// TIA Portal V17 program export: 2 tag tables, 13 data types, 7 data blocks, 53 code blocks (in call order from the OBs), 36 instance data blocks

VAR_GLOBAL   // PLC tag table "Default tag table"
   System_Byte AT %MB1 : Byte;
   FirstScan AT %M1.0 : Bool;
   DiagStatusUpdate AT %M1.1 : Bool;
   Clock_Byte AT %MB0 : Byte;
   Clock_10Hz AT %M0.0 : Bool;
   Clock_5Hz AT %M0.1 : Bool;
   "Clock_2.5Hz" AT %M0.2 : Bool;
   Clock_2Hz AT %M0.3 : Bool;
   "Clock_1.25Hz" AT %M0.4 : Bool;
   Clock_1Hz AT %M0.5 : Bool;
   "Clock_0.625Hz" AT %M0.6 : Bool;
   "Clock_0.5Hz" AT %M0.7 : Bool;
   "System_Byte(1)" AT %MB1 : Byte;
   AlwaysTRUE AT %M1.2 : Bool;
   AlwaysFALSE AT %M1.3 : Bool;
   "System_Byte(2)" AT %MB1 : Byte;
   Tag_1 AT %Q0.6 : Bool;
   Tag_2 AT %M110.0 : Bool;
   Tag_3 AT %M110.1 : Bool;
   Tag_4 AT %MW110 : Word;
END_VAR

VAR_GLOBAL   // PLC tag table "System_Tags"
   pulse_01s AT %M10.0 : Bool;
   pulse_05s AT %M10.1 : Bool;
   pulse_1s AT %M10.2 : Bool;
   pulse_5s AT %M10.3 : Bool;
   pulse_10s AT %M10.4 : Bool;
   pulse_30s AT %M10.5 : Bool;
   pulse_1m AT %M10.6 : Bool;
   pulse_5m AT %M10.7 : Bool;
   pulse_10m AT %M11.0 : Bool;
   pulse_1h AT %M11.2 : Bool;
   TRUE AT %M1.2 : Bool;
   FALSE AT %M1.3 : Bool;
   Hand_DI AT %M12.0 : Bool;
   Hand_DO AT %M12.1 : Bool;
   Hand_AI AT %M12.2 : Bool;
   Hand_AO AT %M12.3 : Bool;
   Hand_M AT %M12.4 : Bool;
   Hand_MD AT %M12.5 : Bool;
   Hand_MDA AT %M12.6 : Bool;
   Hand_V AT %M12.7 : Bool;
   Hand_VD2 AT %M13.0 : Bool;
   Hand_VDA AT %M13.1 : Bool;
   Hand_Any AT %M13.7 : Bool;
   Alm_AI AT %M14.0 : Bool;
   Alm_M AT %M14.1 : Bool;
   Alm_MD AT %M14.2 : Bool;
   Alm_MDA AT %M14.3 : Bool;
   Alm_V AT %M14.4 : Bool;
   Alm_VD2 AT %M14.5 : Bool;
   Alm_VDA AT %M14.6 : Bool;
   Alm_Logick AT %M14.7 : Bool;
   Alm_Any AT %M15.7 : Bool;
   All_Block AT %M2.0 : Bool;
   Reset_All AT %M3.0 : Bool;
   Local_Mode AT %M4.0 : Bool;
   Sim_All AT %M5.0 : Bool;
   AI_Val_1 AT %MB100 : Byte;
   AI_Val_2 AT %MB101 : Byte;
   AI_Value AT %MW100 : Word;
   AO_Val_1 AT %MB102 : Byte;
   AO_Val_2 AT %MB103 : Byte;
   AO_Value AT %MW102 : Word;
   Events AT %MW200 : Word;
   pulse_1_day AT %M11.3 : Bool;
   pulse_1_week AT %M11.4 : Bool;
   pulse_1_month AT %M11.5 : Bool;
   pulse_30m AT %M11.1 : Bool;
   pulse_s1 AT %M11.6 : Bool;
   pulse_s2 AT %M11.7 : Bool;
   Hand_Low AT %M13.5 : Bool;
   Hand_High AT %M13.6 : Bool;
   Reset_Hand AT %M3.1 : Bool;
   Events_pos AT %MW210 : Word;
   Alarms AT %MW202 : Word;
   Alarms_pos AT %MW212 : Word;
END_VAR

TYPE "CMD"
// stored: IsFailsafeCompliant false
   STRUCT
      Start_A : Bool;   // Автозапуск / Запуск в авторежиме
      Start_M : Bool;   // Ручной - вперёд / Запуск в ручном режиме
      Hand : Bool;   // 0 - авто, 1 - ручной / 0 - Авто, 1 - Ручной
      Local : Bool;   // Локальный
      Lock : Bool;   // Блокировать / Блокировка
      Service : Bool;   // Сервис
      Safety : Bool;   // Безопасность
      Force : Bool;   // Принудительный
      Alarm : Bool;   // Есть авария / Авария
      Reset : Bool;   // Сброс аварий
      Sim : Bool;   // Режим симуляции
      Vector { S7_SetPoint := 'True'} : Bool;   // Выбор направления
      ResetOpTime : Bool;   // Сброс счётчика наработки
      Ready : Bool := true;   // Разрешение дистанционного управления
      reserv : Bool;
   END_STRUCT;
END_TYPE

TYPE "InOut_DO"
// stored: IsFailsafeCompliant false
   STRUCT
      CMD : Struct   // Основные команды / Блок команд
         Hand : Bool;   // 0 - авто, 1 - ручной / 0 - Авто, 1 - Ручной
         Start_A : Bool;   // Автозапуск / Запуск в авторежиме
         Start_M : Bool;   // Ручной - вперёд / Запуск в ручном режиме
         Force : Bool;   // Принудительный
         Lock : Bool;   // Блокировать / Блокировка
         Local : Bool;   // Локальный
         Service : Bool;   // Сервис
         Safety : Bool;   // Безопасность
         Alarm : Bool;   // Есть авария / Авария
         Reset : Bool;   // Сброс аварий
         Sim : Bool;   // Режим симуляции
         Vector : Bool;   // Выбор направления
         Ready : Bool;   // Разрешение дистанционного управления
         Resourse : Bool;
      END_STRUCT;
   END_STRUCT;
END_TYPE

TYPE "In_AI"
// stored: IsFailsafeCompliant false
   STRUCT
      Converter : Struct   // Масштабирование сигнала
         Min_Out { S7_SetPoint := 'True'} : Real;   // Минимальный выходной сигнал
         Max_Out { S7_SetPoint := 'True'} : Real := 100.0;   // Максимальный выходной сигнал
      END_STRUCT;
      SP : Struct   // Уставки аварий
         HH { S7_SetPoint := 'True'} : Real := 90.0;
         H { S7_SetPoint := 'True'} : Real := 85.0;
         L { S7_SetPoint := 'True'} : Real := 15.0;
         LL { S7_SetPoint := 'True'} : Real := 10.0;
      END_STRUCT;
   END_STRUCT;
END_TYPE

TYPE "In_MDA"
// stored: IsFailsafeCompliant false
   STRUCT
      CMD : Struct   // Основные команды / Блок команд
         Hand : Bool;   // 0 - авто, 1 - ручной / 0 - Авто, 1 - Ручной
         Start_A : Bool;   // Автозапуск / Запуск в авторежиме
         Start_M : Bool;   // Ручной - вперёд / Запуск в ручном режиме
         Force : Bool;   // Принудительный
         Lock : Bool;   // Блокировать / Блокировка
         Local : Bool;   // Локальный
         Service : Bool;   // Сервис
         Safety : Bool;   // Безопасность
         Alarm : Bool;   // Есть авария / Авария
         Reset : Bool;   // Сброс аварий
         Sim : Bool;   // Режим симуляции
         Vector : Bool;   // Выбор направления
         Ready : Bool;   // Разрешение дистанционного управления
         Resourse : Bool;
      END_STRUCT;
      T_ON : Int;   // Время запуска/открытия
      T_OFF : Int;   // Время останова/закрытия
      SP_M : Real;   // Задание скорости
      Converter : Struct   // Масштабирование сигнала
         Min_Out { S7_SetPoint := 'True'} : Real;   // Минимальный выходной сигнал
         Max_Out { S7_SetPoint := 'True'} : Real := 100.0;   // Максимальный выходной сигнал
      END_STRUCT;
   END_STRUCT;
END_TYPE

TYPE "In_MD_Z"
// stored: IsFailsafeCompliant false
   STRUCT
      CMD : Struct   // Основные команды / Блок команд
         Hand : Bool;   // 0 - авто, 1 - ручной / 0 - Авто, 1 - Ручной
         Start_A : Bool;   // Автозапуск / Запуск в авторежиме
         Start_M : Bool;   // Ручной - вперёд / Запуск в ручном режиме
         Force : Bool;   // Принудительный
         Lock : Bool;   // Блокировать / Блокировка
         Local : Bool;   // Локальный
         Service : Bool;   // Сервис
         Safety : Bool;   // Безопасность
         Alarm : Bool;   // Есть авария / Авария
         Reset : Bool;   // Сброс аварий
         Sim : Bool;   // Режим симуляции
         Vector : Bool;   // Выбор направления
         Ready : Bool;   // Разрешение дистанционного управления
         Resourse : Bool;
      END_STRUCT;
      T_ON : Int;   // Время запуска/открытия
      T_OFF : Int;   // Время останова/закрытия
   END_STRUCT;
END_TYPE

TYPE "Line_Report"
// stored: IsFailsafeCompliant false
   STRUCT
      RM_1 : Real;   // Расход без разбавления
      RM_2 : Real;   // Расход с разбавлением
      Res_1 : Real;   // Наработка насоса 1, часы
      Res_2 : Real;   // Наработка насоса 2, часы
      D_Mid : Real;   // Средняя доза за сутки
      Flow : Real;   // Общая труба (куда происходит дозация)
      WeekDay : Int;   // День недели
      Day : Int;   // Дата записи
      Month : Int;   // Месяц записи
   END_STRUCT;
END_TYPE

TYPE "Out_AI"
// stored: IsFailsafeCompliant false
   STRUCT
      Result : Real;   // Показания датчика
      Converter : Struct   // Масштабирование сигнала
         Min_Out { S7_SetPoint := 'True'} : Real;   // Минимальный выходной сигнал
         Max_Out { S7_SetPoint := 'True'} : Real := 100.0;   // Максимальный выходной сигнал
      END_STRUCT;
      Alarms : Word;   // Слово аварий
      SP : Struct   // Уставки аварий
         HH { S7_SetPoint := 'True'} : Real := 90.0;
         H { S7_SetPoint := 'True'} : Real := 85.0;
         L { S7_SetPoint := 'True'} : Real := 15.0;
         LL { S7_SetPoint := 'True'} : Real := 10.0;
      END_STRUCT;
   END_STRUCT;
END_TYPE

TYPE "Out_MD"
// stored: IsFailsafeCompliant false
   STRUCT
      CMD : Struct   // Основные команды / Блок команд
         Hand : Bool;   // 0 - авто, 1 - ручной / 0 - Авто, 1 - Ручной
         Start_A : Bool;   // Автозапуск / Запуск в авторежиме
         Start_M : Bool;   // Ручной - вперёд / Запуск в ручном режиме
         Force : Bool;   // Принудительный
         Lock : Bool;   // Блокировать / Блокировка
         Local : Bool;   // Локальный
         Service : Bool;   // Сервис
         Safety : Bool;   // Безопасность
         Alarm : Bool;   // Есть авария / Авария
         Reset : Bool;   // Сброс аварий
         Sim : Bool;   // Режим симуляции
         Vector : Bool;   // Выбор направления
         Ready : Bool;   // Разрешение дистанционного управления
         Resourse : Bool;
      END_STRUCT;
      Status : Int;   // Статус устройства
      T_ON : Int;   // Время запуска/открытия
      T_OFF : Int;   // Время останова/закрытия
      Alarms : Word;   // Слово аварий
      Res_h : DInt;   // Текущая уставка
   END_STRUCT;
END_TYPE

TYPE "Out_MDA"
// stored: IsFailsafeCompliant false
   STRUCT
      CMD : Struct   // Основные команды / Блок команд
         Hand : Bool;   // 0 - авто, 1 - ручной / 0 - Авто, 1 - Ручной
         Start_A : Bool;   // Автозапуск / Запуск в авторежиме
         Start_M : Bool;   // Ручной - вперёд / Запуск в ручном режиме
         Force : Bool;   // Принудительный
         Lock : Bool;   // Блокировать / Блокировка
         Local : Bool;   // Локальный
         Service : Bool;   // Сервис
         Safety : Bool;   // Безопасность
         Alarm : Bool;   // Есть авария / Авария
         Reset : Bool;   // Сброс аварий
         Sim : Bool;   // Режим симуляции
         Vector : Bool;   // Выбор направления
         Ready : Bool;   // Разрешение дистанционного управления
         Resourse : Bool;
      END_STRUCT;
      Status : Int;   // Статус устройства
      T_ON : Int;   // Время запуска/открытия
      T_OFF : Int;   // Время останова/закрытия
      Alarms : Word;   // Слово аварий
      Res_h : DInt;   // Наработка, ч
      SP_M : Real;   // Текущая уставка
      Converter : Struct   // Масштабирование сигнала
         Min_Out { S7_SetPoint := 'True'} : Real;   // Минимальный выходной сигнал
         Max_Out { S7_SetPoint := 'True'} : Real := 100.0;   // Максимальный выходной сигнал
      END_STRUCT;
   END_STRUCT;
END_TYPE

TYPE "Out_Z"
// stored: IsFailsafeCompliant false
   STRUCT
      CMD : Struct   // Основные команды / Блок команд
         Hand : Bool;   // 0 - авто, 1 - ручной / 0 - Авто, 1 - Ручной
         Start_A : Bool;   // Автозапуск / Запуск в авторежиме
         Start_M : Bool;   // Ручной - вперёд / Запуск в ручном режиме
         Force : Bool;   // Принудительный
         Lock : Bool;   // Блокировать / Блокировка
         Local : Bool;   // Локальный
         Service : Bool;   // Сервис
         Safety : Bool;   // Безопасность
         Alarm : Bool;   // Есть авария / Авария
         Reset : Bool;   // Сброс аварий
         Sim : Bool;   // Режим симуляции
         Vector : Bool;   // Выбор направления
         Ready : Bool;   // Разрешение дистанционного управления
         Resourse : Bool;
      END_STRUCT;
      Status : Int;   // Статус устройства
      T_ON : Int;   // Время запуска/открытия
      T_OFF : Int;   // Время останова/закрытия
      Alarms : Word;   // Слово аварий
   END_STRUCT;
END_TYPE

TYPE "PolyMix_Input"
// stored: IsFailsafeCompliant false
   STRUCT
      WatchDog : Int;
      Clock : Bool;
      Start : Bool;   // Команда запуска
      SP_C : Real;   // Уставка концентрации
      Weight : Real;
      res_1 : Real;
      res_2 : Real;
   END_STRUCT;
END_TYPE

TYPE "PolyMix_Output"
// stored: IsFailsafeCompliant false
   STRUCT
      WatchDog : Int;
      Clock : Bool;
      Start : Bool;   // Установка в работе
      LS_1 : Bool;   // РУ-1
      LS_2 : Bool;   // РУ-2
      LS_3 : Bool;   // РУ-3
      LS_4 : Bool;   // РУ-4
      KC_1 : Bool;   // Статус клапана КС-1
      ALLS : Bool;   // Аварийно низкий уровень
      Local : Bool;   // 0 - местный режим, 1 - дистанционный
      LLS : Bool;   // Низкий уровень в полимиксе
      HLS : Bool;   // Высокий уровен в полимиксе
      SP_C : Real;   // Заданная концентрация
      Level : Real;   // Уровень в баке
      Flow : Real;   // Скорость потока
      Weight : Real;
      Mix_1 : Int;   // Статус М1
      Mix_2 : Int;   // Статус М2
      Mix_3 : Int;   // Статус М3
      SD : Int;   // Статус ШД
      DD : Int;   // Статус ЧП
      SH : Int;   // Статус ТШ
      PN : Int;   // Статус ПТ
      Vibro : Int;   // Статус вибратора
      Vent : Int;   // Статус вентилятора
      Messages : Struct   // - Аварийные сообщения
         Flow_Dry_Run : Bool;   // Авария - нет протока КС-1
         Flow_Low : Bool;   // Авария - низкий проток КС-1
         LE_NoChange : Bool;   // Авария - не заполняется бак
         LE_Low : Bool;   // Авария - низкий уровень в баке
         LE_High : Bool;   // Авария - высокий уровень в баке
         LS_Low : Bool;   // Авария - низкий уровень в буфере
         LS_NoProduct : Bool;   // Авария - нет продукта в бункере
         LS_Filter : Bool;   // Авария - полный бункер
         SD_Low : Bool;   // Авария - низкая скорость дозации
         Low_Weight : Bool;   // Авария - мало продукта в бункере
         Link_Error : Bool;   // Предупреждение - нет связи со шкафов дозации
         Alarm : Word;   // Слово аварий для панели
      END_STRUCT;
      Report : "PolyMix_Report";   // Отчёт за вчера
      LE_Alarm { S7_SetPoint := 'True'} : Word;   // Слово аврарий датчика уровня
   END_STRUCT;
END_TYPE

TYPE "PolyMix_Report"
// stored: IsFailsafeCompliant false
   STRUCT
      C : Real;   // Средняя концентрация
      Water : Real;   // Расход воды, литры
      Reagent : Real;   // Расход реагента по дозатору, кг
      Weight : Real;   // Расход реагента по весам, кг
      Dos : Real;   // Число доз
      Res : Real;   // Наработка, часы
      WeekDay : Int;   // День недели
      Day : Int;   // Дата записи
      Month : Int;   // Месяц записи
   END_STRUCT;
END_TYPE

DATA_BLOCK "Comm_Scada"   // DB10
{ S7_Optimized_Access := 'FALSE' }
VERSION : 0.1
// stored: AutoNumber false, DBAccessibleFromOPCUA true, IsOnlyStoredInLoadMemory false, IsWriteProtectedInAS false
   VAR
      Input : Struct
         DI_AllBlock : Bool;   // Аварийный останов
         DI_EZ_1_FB_AHLS : Bool;   // Электролизер 1 (Переполнение поддона)
         DI_Gas_Chanel_1_1 : Bool;   // Загазованность канал 1 (Порог 1)
         DI_Gas_Chanel_1_2 : Bool;   // Загазованность канал 1 (Порог 2)
         DI_Gas_Chanel_2_1 : Bool;   // Загазованность канал 2 (Порог 1)
         DI_Gas_Chanel_2_2 : Bool;   // Загазованность канал 2 (Порог 2)
         DI_ALS_1 : Bool;   // Аварийный уровень 1
         ELZ_Wash : Bool;   // Идет промывка
         KC_1 : Bool;   // Промывка фильтра 1
         KC_2 : Bool;   // Промывка фильтра 2
         ELZ_Local : Bool;
         ELZ_1_Status : Int;   // Статус электролизера
         Pump_1_Status : Int;   // Статус насоса 1
         Pump_2_Status : Int;   // Статус насоса 2
         Pump_ELZ_Status : Int;   // Статус насоса электролизера
         RM_1 : Real;   // Импульсный расходомер
         Line_1_Flow_1 : Real;   // Дозирование гипохлорита линии 1
         Line_2_Flow_1 : Real;   // Дозирование гипохлорита линии 2
         AI_LE_1_Result : Real;   // Датчик уровня
         AI_TE_1_Result : Real;   // Датчик температуры
         ELZ_1_Alarm : Word;   // Слово аварий электролизера
         Pump_1_Alarm : Word;   // Слово аварий насоса 1
         Pump_2_Alarm : Word;   // Слово аварий насоса 2
         Pump_ELZ_Alarm : Word;   // Слово аварий электролизера
         AI_LE_1_Alarm : Word;   // Слово аварий датчика уровня
         AI_TE_1_Alarm : Word;   // Слово аварий датчика температуры
         Logick_Alarm : Word;   // Слово аварий блока логики
      END_STRUCT;
      Output : Struct
         Start_ELZ : Bool;   // Запуск электролизера
         Line_1_Start : Bool;   // Старт линии 1
         Line_2_Start : Bool;   // Старт линии 2
         Line_1_Flow : Real;   // Дозирование гипохлорита линии 1
         Line_2_Flow : Real;   // Дозирование гипохлорита линии 2
      END_STRUCT;
   END_VAR
BEGIN
END_DATA_BLOCK

DATA_BLOCK "DB_Comm"   // DB99
{ S7_Optimized_Access := 'FALSE' }
VERSION : 0.1
// stored: AutoNumber false, DBAccessibleFromOPCUA true, IsOnlyStoredInLoadMemory false, IsWriteProtectedInAS false
   VAR RETAIN
      Input : Struct
         Line : Array[0..7] of Struct   // Линии
            Start : Bool;   // Дистанционный старт линии
            Mode : Bool;   // 0 - без разбавления, 1 - с разбавлением
            D : Real;   // Доза линии
         END_STRUCT;
         Pump : Array[1..10] of Struct   // Насосы
            Reserv : Bool;   // 0 - насос основной, 1 - насос резервный
            Line_Main : Int;   // Главная линия насоса
            Line_Reserve : Int;   // Резервная линия насоса
         END_STRUCT;
         Input_PolyMix_1 : "PolyMix_Input";
         Input_PolyMix_2 : "PolyMix_Input";
         Flow_LSAU_1 : Real := 1314.753;   // м3/ч
         Flow_LSAU_2 : Real := 0.0;
         Reset_All : Bool := FALSE;
         PolyMix_1_Source_BK1 : Bool := FALSE;   // Жидкий полимикс - качает с бака 1
         PolyMix_1_Source_BK2 : Bool := TRUE;   // Жидкий полимикс - качает с бака 2
         L123_S_P1 : Bool := FALSE;   // Линия 1 - работает жидким полимиксом
         L123_S_P2 : Bool := TRUE;   // Линия 1 - работает с сухим полимиксом
         L456_S_P1 : Bool := TRUE;   // Линия 2 - работает жидким полимиксом
         L456_S_P2 : Bool := FALSE;   // Линия 2 - работает с сухим полимиксом
         Income_Start : Bool := FALSE;   // Запуск приёмки коагулянта
         Income_Line : Bool := FALSE;   // Приёмка с машины
         Income_Pump : Bool := TRUE;   // Приёмка с кубиков
         Income_BK1 : Bool := TRUE;   // Приёмка в бак БК 1
         Income_BK2 : Bool := FALSE;   // Приёмка в бак БК 2
         Recirk_BK1_Use : Bool := TRUE;   // Автоматическая рециркуляция БК 1
         Recirk_BK2_Use : Bool := TRUE;   // Автоматическая рециркуляция БК 2
         Recirk_BK1_Start : Bool := FALSE;   // Запуск рецикруляции БК 1
         Recirk_BK2_Start : Bool := FALSE;   // Запуск рецикруляции БК 2
         "word" : Word := 16#0000;
      END_STRUCT;
      Output : Struct
         Line : Array[0..7] of Struct   // Линии
            Start : Bool;   // 0 - линия выкл, 1 - линия в работе
            Mode : Bool;   // 0 - без разбавления, 1 - с разбавлением
            Local : Bool;   // 0 - местный режим, 1 - дистанционный
            KC : Bool;   // 0 - КС закрыт, 1 - КС открыт
            RT : Bool;   // 0 - нет протока на РТ, 1 - есть проток на РТ
            D : Real;   // Текущая уставка Дозы
         END_STRUCT;
         Pump : Array[1..10] of Struct   // Насосы
            Reserv : Bool;   // 0 - насос основной, 1 - насос резервный
            Status : Int;   // Статус насоса
            SP : Real;   // Скорость работы насоса
            Line_Main : Int;   // Главная линия насоса
            Line_Reserv : Int;   // Резервная линия насоса
         END_STRUCT;
         Output_PolyMix_1 : "PolyMix_Output";
         Output_PolyMix_2 : "PolyMix_Output";
         PolyMix_1_Source_BK1 : Bool := FALSE;   // Жидкий полимикс - качает с бака 1
         PolyMix_1_Source_BK2 : Bool := TRUE;   // Жидкий полимикс - качает с бака 2
         L123_S_P1 : Bool := FALSE;   // Линия 1 - работает жидким полимиксом
         L123_S_P2 : Bool := TRUE;   // Линия 1 - работает с сухим полимиксом
         L456_S_P1 : Bool := TRUE;   // Линия 2 - работает жидким полимиксом
         L456_S_P2 : Bool := FALSE;   // Линия 2 - работает с сухим полимиксом
         Any_Alarm : Bool := FALSE;   // Общая авария
         Income_Start : Bool := FALSE;   // Запуск приёмки коагулянта
         Income_Line : Bool := FALSE;   // Приёмка с машины
         Income_Pump : Bool := TRUE;   // Приёмка с кубиков
         Income_BK1 : Bool := TRUE;   // Приёмка в бак БК 1
         Income_BK2 : Bool := FALSE;   // Приёмка в бак БК 2
         Recirk_BK1_Use : Bool := TRUE;   // Автоматическая рециркуляция БК 1
         Recirk_BK2_Use : Bool := TRUE;   // Автоматическая рециркуляция БК 2
         Recirk_BK1_Start : Bool := FALSE;   // Запуск рецикруляции БК 1
         Recirk_BK2_Start : Bool := FALSE;   // Запуск рецикруляции БК 2
         reserv : Word := 16#0000;
      END_STRUCT;
      Time_DTL : DTL := DTL#2020-10-13-13:05:17.729949026;
   END_VAR
BEGIN
   Input.Line[0..7].Start := FALSE;
   Input.Line[0].Mode := FALSE;
   Input.Line[1..6].Mode := TRUE;
   Input.Line[7].Mode := FALSE;
   Input.Line[0].D := 3.0;
   Input.Line[1..2].D := 1.0E-05;
   Input.Line[3].D := 3.0E-05;
   Input.Line[4].D := 4.0E-05;
   Input.Line[5].D := 5.0E-05;
   Input.Line[6].D := 6.0E-05;
   Input.Line[7].D := 0.1;
   Input.Pump[1..7].Reserv := FALSE;
   Input.Pump[8].Reserv := TRUE;
   Input.Pump[9].Reserv := FALSE;
   Input.Pump[10].Reserv := TRUE;
   Input.Pump[1].Line_Main := 1;
   Input.Pump[2].Line_Main := 2;
   Input.Pump[3].Line_Main := 3;
   Input.Pump[4].Line_Main := 4;
   Input.Pump[5].Line_Main := 5;
   Input.Pump[6].Line_Main := 6;
   Input.Pump[7].Line_Main := 7;
   Input.Pump[8].Line_Main := 0;
   Input.Pump[9].Line_Main := 8;
   Input.Pump[10].Line_Main := 0;
   Input.Pump[1..7].Line_Reserve := 0;
   Input.Pump[8].Line_Reserve := 7;
   Input.Pump[9].Line_Reserve := 0;
   Input.Pump[10].Line_Reserve := 8;
   Input.Input_PolyMix_1.WatchDog := 2985;   // Контроль связи 0...1000 раз в секунду
   Input.Input_PolyMix_1.Clock := FALSE;   // Контроль связи 1 Гц
   Input.Input_PolyMix_1.Start := TRUE;
   Input.Input_PolyMix_1.SP_C := 9.0;
   Input.Input_PolyMix_1.Weight := 0.0;   // Внешние данные о весе
   Input.Input_PolyMix_1.res_1 := 0.0;   // Резерв 1
   Input.Input_PolyMix_1.res_2 := 0.0;   // Резерв 2
   Input.Input_PolyMix_2.WatchDog := 2985;   // Контроль связи 0...1000 раз в секунду
   Input.Input_PolyMix_2.Clock := FALSE;   // Контроль связи 1 Гц
   Input.Input_PolyMix_2.Start := FALSE;
   Input.Input_PolyMix_2.SP_C := 5.0;
   Input.Input_PolyMix_2.Weight := 593.0253;   // Внешние данные о весе
   Input.Input_PolyMix_2.res_1 := 0.0;   // Резерв 1
   Input.Input_PolyMix_2.res_2 := 0.0;   // Резерв 2
   Output.Line[0..7].Start := FALSE;
   Output.Line[0].Mode := FALSE;
   Output.Line[1..6].Mode := TRUE;
   Output.Line[7].Mode := FALSE;
   Output.Line[0].Local := FALSE;
   Output.Line[1..6].Local := TRUE;
   Output.Line[7].Local := FALSE;
   Output.Line[0..7].KC := FALSE;
   Output.Line[0..7].RT := FALSE;
   Output.Line[0].D := 3.0;
   Output.Line[1..2].D := 1.0E-05;
   Output.Line[3].D := 3.0E-05;
   Output.Line[4].D := 4.0E-05;
   Output.Line[5].D := 5.0E-05;
   Output.Line[6].D := 6.0E-05;
   Output.Line[7].D := 0.1;
   Output.Pump[1..7].Reserv := FALSE;
   Output.Pump[8].Reserv := TRUE;
   Output.Pump[9].Reserv := FALSE;
   Output.Pump[10].Reserv := TRUE;
   Output.Pump[1..10].Status := 0;
   Output.Pump[1..10].SP := 0.0;
   Output.Pump[1].Line_Main := 1;
   Output.Pump[2].Line_Main := 2;
   Output.Pump[3].Line_Main := 3;
   Output.Pump[4].Line_Main := 4;
   Output.Pump[5].Line_Main := 5;
   Output.Pump[6].Line_Main := 6;
   Output.Pump[7].Line_Main := 7;
   Output.Pump[8].Line_Main := 0;
   Output.Pump[9].Line_Main := 8;
   Output.Pump[10].Line_Main := 0;
   Output.Pump[1..7].Line_Reserv := 0;
   Output.Pump[8].Line_Reserv := 7;
   Output.Pump[9].Line_Reserv := 0;
   Output.Pump[10].Line_Reserv := 8;
   Output.Output_PolyMix_1.WatchDog := 182;   // Контроль связи 0...1000 раз в секунду
   Output.Output_PolyMix_1.Clock := TRUE;   // Контроль связи 1 Гц
   Output.Output_PolyMix_1.Start := TRUE;
   Output.Output_PolyMix_1.LS_1 := FALSE;
   Output.Output_PolyMix_1.LS_2 := FALSE;
   Output.Output_PolyMix_1.LS_3 := FALSE;
   Output.Output_PolyMix_1.LS_4 := FALSE;
   Output.Output_PolyMix_1.KC_1 := FALSE;
   Output.Output_PolyMix_1.ALLS := FALSE;
   Output.Output_PolyMix_1.Local := FALSE;
   Output.Output_PolyMix_1.LLS := FALSE;
   Output.Output_PolyMix_1.HLS := TRUE;
   Output.Output_PolyMix_1.SP_C := 9.0;
   Output.Output_PolyMix_1.Level := 985.9791;
   Output.Output_PolyMix_1.Flow := 0.0;
   Output.Output_PolyMix_1.Weight := 0.0;   // Внешние данные о весе
   Output.Output_PolyMix_1.Mix_1 := 0;
   Output.Output_PolyMix_1.Mix_2 := 0;
   Output.Output_PolyMix_1.Mix_3 := 0;
   Output.Output_PolyMix_1.SD := 0;
   Output.Output_PolyMix_1.DD := 0;
   Output.Output_PolyMix_1.SH := 0;
   Output.Output_PolyMix_1.PN := 0;
   Output.Output_PolyMix_1.Vibro := 0;
   Output.Output_PolyMix_1.Vent := 0;
   Output.Output_PolyMix_1.Messages.Flow_Dry_Run := FALSE;
   Output.Output_PolyMix_1.Messages.Flow_Low := FALSE;
   Output.Output_PolyMix_1.Messages.LE_NoChange := FALSE;
   Output.Output_PolyMix_1.Messages.LE_Low := FALSE;
   Output.Output_PolyMix_1.Messages.LE_High := FALSE;
   Output.Output_PolyMix_1.Messages.LS_Low := FALSE;
   Output.Output_PolyMix_1.Messages.LS_NoProduct := FALSE;
   Output.Output_PolyMix_1.Messages.LS_Filter := FALSE;
   Output.Output_PolyMix_1.Messages.SD_Low := FALSE;
   Output.Output_PolyMix_1.Messages.Low_Weight := FALSE;
   Output.Output_PolyMix_1.Messages.Link_Error := FALSE;
   Output.Output_PolyMix_1.Messages.Alarm := 16#0000;
   Output.Output_PolyMix_1.Report.C := 0.0;
   Output.Output_PolyMix_1.Report.Water := 0.0;
   Output.Output_PolyMix_1.Report.Reagent := 0.0;
   Output.Output_PolyMix_1.Report.Weight := 0.0;
   Output.Output_PolyMix_1.Report.Dos := 0.0;
   Output.Output_PolyMix_1.Report.Res := 0.0;
   Output.Output_PolyMix_1.Report.WeekDay := 2;
   Output.Output_PolyMix_1.Report.Day := 12;
   Output.Output_PolyMix_1.Report.Month := 10;
   Output.Output_PolyMix_1.LE_Alarm := 16#0000;
   Output.Output_PolyMix_2.WatchDog := 182;   // Контроль связи 0...1000 раз в секунду
   Output.Output_PolyMix_2.Clock := TRUE;   // Контроль связи 1 Гц
   Output.Output_PolyMix_2.Start := FALSE;
   Output.Output_PolyMix_2.LS_1 := FALSE;
   Output.Output_PolyMix_2.LS_2 := TRUE;
   Output.Output_PolyMix_2.LS_3 := FALSE;
   Output.Output_PolyMix_2.LS_4 := FALSE;
   Output.Output_PolyMix_2.KC_1 := FALSE;
   Output.Output_PolyMix_2.ALLS := FALSE;
   Output.Output_PolyMix_2.Local := FALSE;
   Output.Output_PolyMix_2.LLS := FALSE;
   Output.Output_PolyMix_2.HLS := TRUE;
   Output.Output_PolyMix_2.SP_C := 5.0;
   Output.Output_PolyMix_2.Level := 916.5723;
   Output.Output_PolyMix_2.Flow := 0.0;
   Output.Output_PolyMix_2.Weight := 593.0253;   // Внешние данные о весе
   Output.Output_PolyMix_2.Mix_1 := 1;
   Output.Output_PolyMix_2.Mix_2 := 1;
   Output.Output_PolyMix_2.Mix_3 := 1;
   Output.Output_PolyMix_2.SD := 0;
   Output.Output_PolyMix_2.DD := 0;
   Output.Output_PolyMix_2.SH := 0;
   Output.Output_PolyMix_2.PN := 0;
   Output.Output_PolyMix_2.Vibro := 0;
   Output.Output_PolyMix_2.Vent := 0;
   Output.Output_PolyMix_2.Messages.Flow_Dry_Run := FALSE;
   Output.Output_PolyMix_2.Messages.Flow_Low := FALSE;
   Output.Output_PolyMix_2.Messages.LE_NoChange := FALSE;
   Output.Output_PolyMix_2.Messages.LE_Low := FALSE;
   Output.Output_PolyMix_2.Messages.LE_High := FALSE;
   Output.Output_PolyMix_2.Messages.LS_Low := FALSE;
   Output.Output_PolyMix_2.Messages.LS_NoProduct := FALSE;
   Output.Output_PolyMix_2.Messages.LS_Filter := FALSE;
   Output.Output_PolyMix_2.Messages.SD_Low := FALSE;
   Output.Output_PolyMix_2.Messages.Low_Weight := FALSE;
   Output.Output_PolyMix_2.Messages.Link_Error := FALSE;
   Output.Output_PolyMix_2.Messages.Alarm := 16#0000;
   Output.Output_PolyMix_2.Report.C := 5.0;
   Output.Output_PolyMix_2.Report.Water := 1926.197;
   Output.Output_PolyMix_2.Report.Reagent := 321.0332;
   Output.Output_PolyMix_2.Report.Weight := 0.0;
   Output.Output_PolyMix_2.Report.Dos := 10.0;
   Output.Output_PolyMix_2.Report.Res := 0.0;
   Output.Output_PolyMix_2.Report.WeekDay := 2;
   Output.Output_PolyMix_2.Report.Day := 12;
   Output.Output_PolyMix_2.Report.Month := 10;
   Output.Output_PolyMix_2.LE_Alarm := 16#0000;
END_DATA_BLOCK

DATA_BLOCK "DB_IN"   // DB101
{ S7_Optimized_Access := 'FALSE' }
VERSION : 0.1
// stored: AutoNumber false, DBAccessibleFromOPCUA true, IsOnlyStoredInLoadMemory false, IsWriteProtectedInAS false
   VAR RETAIN
      PolyMix_1 : Struct
         Start : Bool := FALSE;
         SP_C : Real := 0.0;
      END_STRUCT;
      PolyMix_2 : Struct
         Start : Bool := FALSE;
         SP_C : Real := 0.0;
      END_STRUCT;
      AI_FT_007 : "In_AI";
      AI_FT_008 { S7_SetPoint := 'True'} : "In_AI";
      AI_FT_009 { S7_SetPoint := 'True'} : "In_AI";
      AI_FT_010 { S7_SetPoint := 'True'} : "In_AI";
      AI_LT_014 { S7_SetPoint := 'True'} : "In_AI";
      AI_LT_015 { S7_SetPoint := 'True'} : "In_AI";
      AI_LT_016 { S7_SetPoint := 'True'} : "In_AI";
      AI_LT_019 { S7_SetPoint := 'True'} : "In_AI";
      AI_PT_001 { S7_SetPoint := 'True'} : "In_AI";
      AI_PT_002 { S7_SetPoint := 'True'} : "In_AI";
      AI_PT_003 { S7_SetPoint := 'True'} : "In_AI";
      AI_PT_004 { S7_SetPoint := 'True'} : "In_AI";
      AI_PT_005 { S7_SetPoint := 'True'} : "In_AI";
      AI_PT_006 { S7_SetPoint := 'True'} : "In_AI";
      Z_GVM_020 { S7_SetPoint := 'True'} : "In_MD_Z";
      Z_GVM_021 { S7_SetPoint := 'True'} : "In_MD_Z";
      Z_GVM_022 { S7_SetPoint := 'True'} : "In_MD_Z";
      Z_GCM_023 { S7_SetPoint := 'True'} : "In_MD_Z";
      Z_GCM_024 { S7_SetPoint := 'True'} : "In_MD_Z";
      Z_GCM_025 { S7_SetPoint := 'True'} : "In_MD_Z";
      XVS_026 { S7_SetPoint := 'True'} : "InOut_DO";
      XVS_027 { S7_SetPoint := 'True'} : "InOut_DO";
      XVS_028 { S7_SetPoint := 'True'} : "InOut_DO";
      XVS_029 { S7_SetPoint := 'True'} : "InOut_DO";
      XVS_030 { S7_SetPoint := 'True'} : "InOut_DO";
      XVS_031 { S7_SetPoint := 'True'} : "InOut_DO";
      XVS_032 { S7_SetPoint := 'True'} : "InOut_DO";
      XVS_033 { S7_SetPoint := 'True'} : "InOut_DO";
      XVS_034 { S7_SetPoint := 'True'} : "InOut_DO";
      M6_M_K_1_1 { S7_SetPoint := 'True'} : "In_MD_Z";
      M7_M_K_1_2 { S7_SetPoint := 'True'} : "In_MD_Z";
      M8_M_K_1_3 { S7_SetPoint := 'True'} : "In_MD_Z";
      M11_M_K_2_1 { S7_SetPoint := 'True'} : "In_MD_Z";
      M12_M_K_2_2 { S7_SetPoint := 'True'} : "In_MD_Z";
      M13_M_K_2_3 { S7_SetPoint := 'True'} : "In_MD_Z";
      M9_SD { S7_SetPoint := 'True'} : "In_MDA";
      M10_Vibro_1 { S7_SetPoint := 'True'} : "In_MD_Z";
      M1_BK_1 { S7_SetPoint := 'True'} : "In_MDA";
      M2_KK_1_1 { S7_SetPoint := 'True'} : "In_MDA";
      M3_KK_1_2 { S7_SetPoint := 'True'} : "In_MDA";
      M4_ND_KK_1_1 { S7_SetPoint := 'True'} : "In_MDA";
      M5_ND_KK_1_2 { S7_SetPoint := 'True'} : "In_MDA";
      M14_ND_K_1_1 { S7_SetPoint := 'True'} : "In_MDA";
      M15_ND_K_1_2 { S7_SetPoint := 'True'} : "In_MDA";
      M16_ND_K_1_3 { S7_SetPoint := 'True'} : "In_MDA";
      M17_ND_K_2_1 { S7_SetPoint := 'True'} : "In_MDA";
      M18_ND_K_2_2 { S7_SetPoint := 'True'} : "In_MDA";
      M19_ND_K_2_3 : "In_MDA";
      XVS_035 { S7_SetPoint := 'True'} : "InOut_DO";
      XVS_036 { S7_SetPoint := 'True'} : "InOut_DO";
      gsm3_PolyMix_1 { S7_SetPoint := 'True'} : Real := 1.09;
      gsm3_PolyMix_2 : Real := 1.072;
      F1_Clean_CMD : Bool := FALSE;
      F2_Clean_CMD : Bool := FALSE;
      Z_GVM_x { S7_SetPoint := 'True'} : "In_MD_Z";
      res_1 : Word := 16#0000;
      res_2 : Word := 16#0000;
      res_3 : Word := 16#0000;
      res_4 : Word := 16#0000;
      res_5 : Word := 16#0000;
      res_6 : Word := 16#0000;
      res_7 : Word := 16#0000;
      res_8 : Word := 16#0000;
      res_9 : Word := 16#0000;
      res_10 : Word := 16#0000;
      Time_DTL : DTL := DTL#2020-06-25-13:08:09.170187013;
   END_VAR
BEGIN
   AI_FT_007.Converter.Min_Out := 0.0;
   AI_FT_007.Converter.Max_Out := 1000.0;
   AI_FT_007.SP.HH := 320.0;
   AI_FT_007.SP.H := 300.0;
   AI_FT_007.SP.L := 200.0;
   AI_FT_007.SP.LL := 75.0;
   AI_FT_008.Converter.Min_Out := 0.0;
   AI_FT_008.Converter.Max_Out := 100.0;
   AI_FT_008.SP.HH := 100.0;
   AI_FT_008.SP.H := 15.0;
   AI_FT_008.SP.L := 0.5;
   AI_FT_008.SP.LL := -0.1;
   AI_FT_009.Converter.Min_Out := 0.0;
   AI_FT_009.Converter.Max_Out := 100.0;
   AI_FT_009.SP.HH := 30.0;
   AI_FT_009.SP.H := 15.0;
   AI_FT_009.SP.L := 0.5;
   AI_FT_009.SP.LL := -0.1;
   AI_FT_010.Converter.Min_Out := 0.0;
   AI_FT_010.Converter.Max_Out := 100.0;
   AI_FT_010.SP.HH := 50.0;
   AI_FT_010.SP.H := 40.0;
   AI_FT_010.SP.L := 0.5;
   AI_FT_010.SP.LL := -0.5;
   AI_LT_014.Converter.Min_Out := 0.0;
   AI_LT_014.Converter.Max_Out := 2605.0;
   AI_LT_014.SP.HH := 2400.0;
   AI_LT_014.SP.H := 2300.0;
   AI_LT_014.SP.L := 400.0;
   AI_LT_014.SP.LL := 220.0;
   AI_LT_015.Converter.Min_Out := 0.0;
   AI_LT_015.Converter.Max_Out := 2605.0;
   AI_LT_015.SP.HH := 2400.0;
   AI_LT_015.SP.H := 2300.0;
   AI_LT_015.SP.L := 400.0;
   AI_LT_015.SP.LL := 220.0;
   AI_LT_016.Converter.Min_Out := 0.0;
   AI_LT_016.Converter.Max_Out := 1268.0;
   AI_LT_016.SP.HH := 1060.0;
   AI_LT_016.SP.H := 950.0;
   AI_LT_016.SP.L := 250.0;
   AI_LT_016.SP.LL := 120.0;
   AI_LT_019.Converter.Min_Out := 0.0;
   AI_LT_019.Converter.Max_Out := 1268.0;
   AI_LT_019.SP.HH := 1060.0;
   AI_LT_019.SP.H := 950.0;
   AI_LT_019.SP.L := 250.0;
   AI_LT_019.SP.LL := 120.0;
   AI_PT_001.Converter.Min_Out := 0.0;
   AI_PT_001.Converter.Max_Out := 0.6;
   AI_PT_001.SP.HH := 0.35;
   AI_PT_001.SP.H := 0.3;
   AI_PT_001.SP.L := 0.02;
   AI_PT_001.SP.LL := 0.01;
   AI_PT_002.Converter.Min_Out := 0.0;
   AI_PT_002.Converter.Max_Out := 0.6;
   AI_PT_002.SP.HH := 0.35;
   AI_PT_002.SP.H := 0.3;
   AI_PT_002.SP.L := 0.02;
   AI_PT_002.SP.LL := 0.01;
   AI_PT_003.Converter.Min_Out := 0.0;
   AI_PT_003.Converter.Max_Out := 0.6;
   AI_PT_003.SP.HH := 0.35;
   AI_PT_003.SP.H := 0.3;
   AI_PT_003.SP.L := 0.02;
   AI_PT_003.SP.LL := 0.01;
   AI_PT_004.Converter.Min_Out := 0.0;
   AI_PT_004.Converter.Max_Out := 0.6;
   AI_PT_004.SP.HH := 0.35;
   AI_PT_004.SP.H := 0.3;
   AI_PT_004.SP.L := 0.02;
   AI_PT_004.SP.LL := 0.01;
   AI_PT_005.Converter.Min_Out := 0.0;
   AI_PT_005.Converter.Max_Out := 0.6;
   AI_PT_005.SP.HH := 0.35;
   AI_PT_005.SP.H := 0.3;
   AI_PT_005.SP.L := 0.02;
   AI_PT_005.SP.LL := 0.01;
   AI_PT_006.Converter.Min_Out := 0.0;
   AI_PT_006.Converter.Max_Out := 0.6;
   AI_PT_006.SP.HH := 0.35;
   AI_PT_006.SP.H := 0.3;
   AI_PT_006.SP.L := 0.02;
   AI_PT_006.SP.LL := 0.01;
   Z_GVM_020.CMD.Hand := FALSE;
   Z_GVM_020.CMD.Start_A := FALSE;
   Z_GVM_020.CMD.Start_M := FALSE;
   Z_GVM_020.CMD.Force := FALSE;
   Z_GVM_020.CMD.Lock := FALSE;
   Z_GVM_020.CMD.Local := FALSE;
   Z_GVM_020.CMD.Service := FALSE;
   Z_GVM_020.CMD.Safety := FALSE;
   Z_GVM_020.CMD.Alarm := FALSE;
   Z_GVM_020.CMD.Reset := FALSE;
   Z_GVM_020.CMD.Sim := FALSE;
   Z_GVM_020.CMD.Vector := FALSE;
   Z_GVM_020.CMD.Ready := FALSE;
   Z_GVM_020.CMD.Resourse := FALSE;
   Z_GVM_020.T_ON := 12;
   Z_GVM_020.T_OFF := 12;
   Z_GVM_021.CMD.Hand := FALSE;
   Z_GVM_021.CMD.Start_A := FALSE;
   Z_GVM_021.CMD.Start_M := FALSE;
   Z_GVM_021.CMD.Force := FALSE;
   Z_GVM_021.CMD.Lock := FALSE;
   Z_GVM_021.CMD.Local := FALSE;
   Z_GVM_021.CMD.Service := FALSE;
   Z_GVM_021.CMD.Safety := FALSE;
   Z_GVM_021.CMD.Alarm := FALSE;
   Z_GVM_021.CMD.Reset := FALSE;
   Z_GVM_021.CMD.Sim := FALSE;
   Z_GVM_021.CMD.Vector := FALSE;
   Z_GVM_021.CMD.Ready := FALSE;
   Z_GVM_021.CMD.Resourse := FALSE;
   Z_GVM_021.T_ON := 12;
   Z_GVM_021.T_OFF := 12;
   Z_GVM_022.CMD.Hand := FALSE;
   Z_GVM_022.CMD.Start_A := FALSE;
   Z_GVM_022.CMD.Start_M := FALSE;
   Z_GVM_022.CMD.Force := FALSE;
   Z_GVM_022.CMD.Lock := FALSE;
   Z_GVM_022.CMD.Local := FALSE;
   Z_GVM_022.CMD.Service := FALSE;
   Z_GVM_022.CMD.Safety := FALSE;
   Z_GVM_022.CMD.Alarm := FALSE;
   Z_GVM_022.CMD.Reset := FALSE;
   Z_GVM_022.CMD.Sim := FALSE;
   Z_GVM_022.CMD.Vector := FALSE;
   Z_GVM_022.CMD.Ready := FALSE;
   Z_GVM_022.CMD.Resourse := FALSE;
   Z_GVM_022.T_ON := 12;
   Z_GVM_022.T_OFF := 12;
   Z_GCM_023.CMD.Hand := FALSE;
   Z_GCM_023.CMD.Start_A := FALSE;
   Z_GCM_023.CMD.Start_M := FALSE;
   Z_GCM_023.CMD.Force := FALSE;
   Z_GCM_023.CMD.Lock := FALSE;
   Z_GCM_023.CMD.Local := FALSE;
   Z_GCM_023.CMD.Service := FALSE;
   Z_GCM_023.CMD.Safety := FALSE;
   Z_GCM_023.CMD.Alarm := FALSE;
   Z_GCM_023.CMD.Reset := FALSE;
   Z_GCM_023.CMD.Sim := FALSE;
   Z_GCM_023.CMD.Vector := FALSE;
   Z_GCM_023.CMD.Ready := FALSE;
   Z_GCM_023.CMD.Resourse := FALSE;
   Z_GCM_023.T_ON := 12;
   Z_GCM_023.T_OFF := 12;
   Z_GCM_024.CMD.Hand := FALSE;
   Z_GCM_024.CMD.Start_A := FALSE;
   Z_GCM_024.CMD.Start_M := FALSE;
   Z_GCM_024.CMD.Force := FALSE;
   Z_GCM_024.CMD.Lock := FALSE;
   Z_GCM_024.CMD.Local := FALSE;
   Z_GCM_024.CMD.Service := FALSE;
   Z_GCM_024.CMD.Safety := FALSE;
   Z_GCM_024.CMD.Alarm := FALSE;
   Z_GCM_024.CMD.Reset := FALSE;
   Z_GCM_024.CMD.Sim := FALSE;
   Z_GCM_024.CMD.Vector := FALSE;
   Z_GCM_024.CMD.Ready := FALSE;
   Z_GCM_024.CMD.Resourse := FALSE;
   Z_GCM_024.T_ON := 12;
   Z_GCM_024.T_OFF := 12;
   Z_GCM_025.CMD.Hand := FALSE;
   Z_GCM_025.CMD.Start_A := FALSE;
   Z_GCM_025.CMD.Start_M := FALSE;
   Z_GCM_025.CMD.Force := FALSE;
   Z_GCM_025.CMD.Lock := FALSE;
   Z_GCM_025.CMD.Local := FALSE;
   Z_GCM_025.CMD.Service := FALSE;
   Z_GCM_025.CMD.Safety := FALSE;
   Z_GCM_025.CMD.Alarm := FALSE;
   Z_GCM_025.CMD.Reset := FALSE;
   Z_GCM_025.CMD.Sim := FALSE;
   Z_GCM_025.CMD.Vector := FALSE;
   Z_GCM_025.CMD.Ready := FALSE;
   Z_GCM_025.CMD.Resourse := FALSE;
   Z_GCM_025.T_ON := 12;
   Z_GCM_025.T_OFF := 12;
   XVS_026.CMD.Hand := FALSE;
   XVS_026.CMD.Start_A := FALSE;
   XVS_026.CMD.Start_M := FALSE;
   XVS_026.CMD.Force := FALSE;
   XVS_026.CMD.Lock := FALSE;
   XVS_026.CMD.Local := FALSE;
   XVS_026.CMD.Service := FALSE;
   XVS_026.CMD.Safety := FALSE;
   XVS_026.CMD.Alarm := FALSE;
   XVS_026.CMD.Reset := FALSE;
   XVS_026.CMD.Sim := FALSE;
   XVS_026.CMD.Vector := FALSE;
   XVS_026.CMD.Ready := FALSE;
   XVS_026.CMD.Resourse := FALSE;
   XVS_027.CMD.Hand := FALSE;
   XVS_027.CMD.Start_A := FALSE;
   XVS_027.CMD.Start_M := FALSE;
   XVS_027.CMD.Force := FALSE;
   XVS_027.CMD.Lock := FALSE;
   XVS_027.CMD.Local := FALSE;
   XVS_027.CMD.Service := FALSE;
   XVS_027.CMD.Safety := FALSE;
   XVS_027.CMD.Alarm := FALSE;
   XVS_027.CMD.Reset := FALSE;
   XVS_027.CMD.Sim := FALSE;
   XVS_027.CMD.Vector := FALSE;
   XVS_027.CMD.Ready := FALSE;
   XVS_027.CMD.Resourse := FALSE;
   XVS_028.CMD.Hand := FALSE;
   XVS_028.CMD.Start_A := FALSE;
   XVS_028.CMD.Start_M := FALSE;
   XVS_028.CMD.Force := FALSE;
   XVS_028.CMD.Lock := FALSE;
   XVS_028.CMD.Local := FALSE;
   XVS_028.CMD.Service := FALSE;
   XVS_028.CMD.Safety := FALSE;
   XVS_028.CMD.Alarm := FALSE;
   XVS_028.CMD.Reset := FALSE;
   XVS_028.CMD.Sim := FALSE;
   XVS_028.CMD.Vector := FALSE;
   XVS_028.CMD.Ready := FALSE;
   XVS_028.CMD.Resourse := FALSE;
   XVS_029.CMD.Hand := FALSE;
   XVS_029.CMD.Start_A := FALSE;
   XVS_029.CMD.Start_M := FALSE;
   XVS_029.CMD.Force := FALSE;
   XVS_029.CMD.Lock := FALSE;
   XVS_029.CMD.Local := FALSE;
   XVS_029.CMD.Service := FALSE;
   XVS_029.CMD.Safety := FALSE;
   XVS_029.CMD.Alarm := FALSE;
   XVS_029.CMD.Reset := FALSE;
   XVS_029.CMD.Sim := FALSE;
   XVS_029.CMD.Vector := FALSE;
   XVS_029.CMD.Ready := FALSE;
   XVS_029.CMD.Resourse := FALSE;
   XVS_030.CMD.Hand := FALSE;
   XVS_030.CMD.Start_A := FALSE;
   XVS_030.CMD.Start_M := FALSE;
   XVS_030.CMD.Force := FALSE;
   XVS_030.CMD.Lock := FALSE;
   XVS_030.CMD.Local := FALSE;
   XVS_030.CMD.Service := FALSE;
   XVS_030.CMD.Safety := FALSE;
   XVS_030.CMD.Alarm := FALSE;
   XVS_030.CMD.Reset := FALSE;
   XVS_030.CMD.Sim := FALSE;
   XVS_030.CMD.Vector := FALSE;
   XVS_030.CMD.Ready := FALSE;
   XVS_030.CMD.Resourse := FALSE;
   XVS_031.CMD.Hand := FALSE;
   XVS_031.CMD.Start_A := FALSE;
   XVS_031.CMD.Start_M := FALSE;
   XVS_031.CMD.Force := FALSE;
   XVS_031.CMD.Lock := FALSE;
   XVS_031.CMD.Local := FALSE;
   XVS_031.CMD.Service := FALSE;
   XVS_031.CMD.Safety := FALSE;
   XVS_031.CMD.Alarm := FALSE;
   XVS_031.CMD.Reset := FALSE;
   XVS_031.CMD.Sim := FALSE;
   XVS_031.CMD.Vector := FALSE;
   XVS_031.CMD.Ready := FALSE;
   XVS_031.CMD.Resourse := FALSE;
   XVS_032.CMD.Hand := FALSE;
   XVS_032.CMD.Start_A := FALSE;
   XVS_032.CMD.Start_M := FALSE;
   XVS_032.CMD.Force := FALSE;
   XVS_032.CMD.Lock := FALSE;
   XVS_032.CMD.Local := FALSE;
   XVS_032.CMD.Service := FALSE;
   XVS_032.CMD.Safety := FALSE;
   XVS_032.CMD.Alarm := FALSE;
   XVS_032.CMD.Reset := FALSE;
   XVS_032.CMD.Sim := FALSE;
   XVS_032.CMD.Vector := FALSE;
   XVS_032.CMD.Ready := FALSE;
   XVS_032.CMD.Resourse := FALSE;
   XVS_033.CMD.Hand := FALSE;
   XVS_033.CMD.Start_A := FALSE;
   XVS_033.CMD.Start_M := FALSE;
   XVS_033.CMD.Force := FALSE;
   XVS_033.CMD.Lock := FALSE;
   XVS_033.CMD.Local := FALSE;
   XVS_033.CMD.Service := FALSE;
   XVS_033.CMD.Safety := FALSE;
   XVS_033.CMD.Alarm := FALSE;
   XVS_033.CMD.Reset := FALSE;
   XVS_033.CMD.Sim := FALSE;
   XVS_033.CMD.Vector := FALSE;
   XVS_033.CMD.Ready := FALSE;
   XVS_033.CMD.Resourse := FALSE;
   XVS_034.CMD.Hand := FALSE;
   XVS_034.CMD.Start_A := FALSE;
   XVS_034.CMD.Start_M := FALSE;
   XVS_034.CMD.Force := FALSE;
   XVS_034.CMD.Lock := FALSE;
   XVS_034.CMD.Local := FALSE;
   XVS_034.CMD.Service := FALSE;
   XVS_034.CMD.Safety := FALSE;
   XVS_034.CMD.Alarm := FALSE;
   XVS_034.CMD.Reset := FALSE;
   XVS_034.CMD.Sim := FALSE;
   XVS_034.CMD.Vector := FALSE;
   XVS_034.CMD.Ready := FALSE;
   XVS_034.CMD.Resourse := FALSE;
   M6_M_K_1_1.CMD.Hand := FALSE;
   M6_M_K_1_1.CMD.Start_A := TRUE;
   M6_M_K_1_1.CMD.Start_M := TRUE;
   M6_M_K_1_1.CMD.Force := FALSE;
   M6_M_K_1_1.CMD.Lock := FALSE;
   M6_M_K_1_1.CMD.Local := FALSE;
   M6_M_K_1_1.CMD.Service := FALSE;
   M6_M_K_1_1.CMD.Safety := FALSE;
   M6_M_K_1_1.CMD.Alarm := FALSE;
   M6_M_K_1_1.CMD.Reset := FALSE;
   M6_M_K_1_1.CMD.Sim := FALSE;
   M6_M_K_1_1.CMD.Vector := FALSE;
   M6_M_K_1_1.CMD.Ready := FALSE;
   M6_M_K_1_1.CMD.Resourse := FALSE;
   M6_M_K_1_1.T_ON := 2;
   M6_M_K_1_1.T_OFF := 2;
   M7_M_K_1_2.CMD.Hand := FALSE;
   M7_M_K_1_2.CMD.Start_A := TRUE;
   M7_M_K_1_2.CMD.Start_M := TRUE;
   M7_M_K_1_2.CMD.Force := FALSE;
   M7_M_K_1_2.CMD.Lock := FALSE;
   M7_M_K_1_2.CMD.Local := FALSE;
   M7_M_K_1_2.CMD.Service := FALSE;
   M7_M_K_1_2.CMD.Safety := FALSE;
   M7_M_K_1_2.CMD.Alarm := FALSE;
   M7_M_K_1_2.CMD.Reset := FALSE;
   M7_M_K_1_2.CMD.Sim := FALSE;
   M7_M_K_1_2.CMD.Vector := FALSE;
   M7_M_K_1_2.CMD.Ready := FALSE;
   M7_M_K_1_2.CMD.Resourse := FALSE;
   M7_M_K_1_2.T_ON := 2;
   M7_M_K_1_2.T_OFF := 2;
   M8_M_K_1_3.CMD.Hand := FALSE;
   M8_M_K_1_3.CMD.Start_A := TRUE;
   M8_M_K_1_3.CMD.Start_M := TRUE;
   M8_M_K_1_3.CMD.Force := FALSE;
   M8_M_K_1_3.CMD.Lock := FALSE;
   M8_M_K_1_3.CMD.Local := FALSE;
   M8_M_K_1_3.CMD.Service := FALSE;
   M8_M_K_1_3.CMD.Safety := FALSE;
   M8_M_K_1_3.CMD.Alarm := FALSE;
   M8_M_K_1_3.CMD.Reset := FALSE;
   M8_M_K_1_3.CMD.Sim := FALSE;
   M8_M_K_1_3.CMD.Vector := FALSE;
   M8_M_K_1_3.CMD.Ready := FALSE;
   M8_M_K_1_3.CMD.Resourse := FALSE;
   M8_M_K_1_3.T_ON := 2;
   M8_M_K_1_3.T_OFF := 2;
   M11_M_K_2_1.CMD.Hand := FALSE;
   M11_M_K_2_1.CMD.Start_A := FALSE;
   M11_M_K_2_1.CMD.Start_M := FALSE;
   M11_M_K_2_1.CMD.Force := FALSE;
   M11_M_K_2_1.CMD.Lock := FALSE;
   M11_M_K_2_1.CMD.Local := FALSE;
   M11_M_K_2_1.CMD.Service := FALSE;
   M11_M_K_2_1.CMD.Safety := FALSE;
   M11_M_K_2_1.CMD.Alarm := FALSE;
   M11_M_K_2_1.CMD.Reset := FALSE;
   M11_M_K_2_1.CMD.Sim := FALSE;
   M11_M_K_2_1.CMD.Vector := FALSE;
   M11_M_K_2_1.CMD.Ready := FALSE;
   M11_M_K_2_1.CMD.Resourse := FALSE;
   M11_M_K_2_1.T_ON := 2;
   M11_M_K_2_1.T_OFF := 2;
   M12_M_K_2_2.CMD.Hand := FALSE;
   M12_M_K_2_2.CMD.Start_A := FALSE;
   M12_M_K_2_2.CMD.Start_M := FALSE;
   M12_M_K_2_2.CMD.Force := FALSE;
   M12_M_K_2_2.CMD.Lock := FALSE;
   M12_M_K_2_2.CMD.Local := FALSE;
   M12_M_K_2_2.CMD.Service := FALSE;
   M12_M_K_2_2.CMD.Safety := FALSE;
   M12_M_K_2_2.CMD.Alarm := FALSE;
   M12_M_K_2_2.CMD.Reset := FALSE;
   M12_M_K_2_2.CMD.Sim := FALSE;
   M12_M_K_2_2.CMD.Vector := FALSE;
   M12_M_K_2_2.CMD.Ready := FALSE;
   M12_M_K_2_2.CMD.Resourse := FALSE;
   M12_M_K_2_2.T_ON := 2;
   M12_M_K_2_2.T_OFF := 2;
   M13_M_K_2_3.CMD.Hand := FALSE;
   M13_M_K_2_3.CMD.Start_A := FALSE;
   M13_M_K_2_3.CMD.Start_M := FALSE;
   M13_M_K_2_3.CMD.Force := FALSE;
   M13_M_K_2_3.CMD.Lock := FALSE;
   M13_M_K_2_3.CMD.Local := FALSE;
   M13_M_K_2_3.CMD.Service := FALSE;
   M13_M_K_2_3.CMD.Safety := FALSE;
   M13_M_K_2_3.CMD.Alarm := FALSE;
   M13_M_K_2_3.CMD.Reset := FALSE;
   M13_M_K_2_3.CMD.Sim := FALSE;
   M13_M_K_2_3.CMD.Vector := FALSE;
   M13_M_K_2_3.CMD.Ready := FALSE;
   M13_M_K_2_3.CMD.Resourse := FALSE;
   M13_M_K_2_3.T_ON := 2;
   M13_M_K_2_3.T_OFF := 2;
   M9_SD.CMD.Hand := FALSE;
   M9_SD.CMD.Start_A := FALSE;
   M9_SD.CMD.Start_M := FALSE;
   M9_SD.CMD.Force := FALSE;
   M9_SD.CMD.Lock := FALSE;
   M9_SD.CMD.Local := FALSE;
   M9_SD.CMD.Service := FALSE;
   M9_SD.CMD.Safety := FALSE;
   M9_SD.CMD.Alarm := FALSE;
   M9_SD.CMD.Reset := FALSE;
   M9_SD.CMD.Sim := FALSE;
   M9_SD.CMD.Vector := FALSE;
   M9_SD.CMD.Ready := FALSE;
   M9_SD.CMD.Resourse := FALSE;
   M9_SD.T_ON := 2;
   M9_SD.T_OFF := 2;
   M9_SD.SP_M := 0.0;
   M9_SD.Converter.Min_Out := 0.0;
   M9_SD.Converter.Max_Out := 100.0;
   M10_Vibro_1.CMD.Hand := FALSE;
   M10_Vibro_1.CMD.Start_A := FALSE;
   M10_Vibro_1.CMD.Start_M := FALSE;
   M10_Vibro_1.CMD.Force := FALSE;
   M10_Vibro_1.CMD.Lock := FALSE;
   M10_Vibro_1.CMD.Local := FALSE;
   M10_Vibro_1.CMD.Service := FALSE;
   M10_Vibro_1.CMD.Safety := FALSE;
   M10_Vibro_1.CMD.Alarm := FALSE;
   M10_Vibro_1.CMD.Reset := FALSE;
   M10_Vibro_1.CMD.Sim := FALSE;
   M10_Vibro_1.CMD.Vector := FALSE;
   M10_Vibro_1.CMD.Ready := FALSE;
   M10_Vibro_1.CMD.Resourse := FALSE;
   M10_Vibro_1.T_ON := 2;
   M10_Vibro_1.T_OFF := 2;
   M1_BK_1.CMD.Hand := FALSE;
   M1_BK_1.CMD.Start_A := FALSE;
   M1_BK_1.CMD.Start_M := FALSE;
   M1_BK_1.CMD.Force := FALSE;
   M1_BK_1.CMD.Lock := FALSE;
   M1_BK_1.CMD.Local := FALSE;
   M1_BK_1.CMD.Service := FALSE;
   M1_BK_1.CMD.Safety := FALSE;
   M1_BK_1.CMD.Alarm := FALSE;
   M1_BK_1.CMD.Reset := FALSE;
   M1_BK_1.CMD.Sim := FALSE;
   M1_BK_1.CMD.Vector := FALSE;
   M1_BK_1.CMD.Ready := FALSE;
   M1_BK_1.CMD.Resourse := FALSE;
   M1_BK_1.T_ON := 2;
   M1_BK_1.T_OFF := 2;
   M1_BK_1.SP_M := 0.0;
   M1_BK_1.Converter.Min_Out := 0.0;
   M1_BK_1.Converter.Max_Out := 0.0;
   M2_KK_1_1.CMD.Hand := FALSE;
   M2_KK_1_1.CMD.Start_A := FALSE;
   M2_KK_1_1.CMD.Start_M := FALSE;
   M2_KK_1_1.CMD.Force := FALSE;
   M2_KK_1_1.CMD.Lock := FALSE;
   M2_KK_1_1.CMD.Local := FALSE;
   M2_KK_1_1.CMD.Service := FALSE;
   M2_KK_1_1.CMD.Safety := FALSE;
   M2_KK_1_1.CMD.Alarm := FALSE;
   M2_KK_1_1.CMD.Reset := FALSE;
   M2_KK_1_1.CMD.Sim := FALSE;
   M2_KK_1_1.CMD.Vector := FALSE;
   M2_KK_1_1.CMD.Ready := FALSE;
   M2_KK_1_1.CMD.Resourse := FALSE;
   M2_KK_1_1.T_ON := 2;
   M2_KK_1_1.T_OFF := 2;
   M2_KK_1_1.SP_M := 0.0;
   M2_KK_1_1.Converter.Min_Out := 0.0;
   M2_KK_1_1.Converter.Max_Out := 0.0;
   M3_KK_1_2.CMD.Hand := FALSE;
   M3_KK_1_2.CMD.Start_A := FALSE;
   M3_KK_1_2.CMD.Start_M := FALSE;
   M3_KK_1_2.CMD.Force := FALSE;
   M3_KK_1_2.CMD.Lock := FALSE;
   M3_KK_1_2.CMD.Local := FALSE;
   M3_KK_1_2.CMD.Service := FALSE;
   M3_KK_1_2.CMD.Safety := FALSE;
   M3_KK_1_2.CMD.Alarm := FALSE;
   M3_KK_1_2.CMD.Reset := FALSE;
   M3_KK_1_2.CMD.Sim := FALSE;
   M3_KK_1_2.CMD.Vector := FALSE;
   M3_KK_1_2.CMD.Ready := FALSE;
   M3_KK_1_2.CMD.Resourse := FALSE;
   M3_KK_1_2.T_ON := 2;
   M3_KK_1_2.T_OFF := 2;
   M3_KK_1_2.SP_M := 0.0;
   M3_KK_1_2.Converter.Min_Out := 0.0;
   M3_KK_1_2.Converter.Max_Out := 0.0;
   M4_ND_KK_1_1.CMD.Hand := FALSE;
   M4_ND_KK_1_1.CMD.Start_A := FALSE;
   M4_ND_KK_1_1.CMD.Start_M := FALSE;
   M4_ND_KK_1_1.CMD.Force := FALSE;
   M4_ND_KK_1_1.CMD.Lock := FALSE;
   M4_ND_KK_1_1.CMD.Local := FALSE;
   M4_ND_KK_1_1.CMD.Service := FALSE;
   M4_ND_KK_1_1.CMD.Safety := FALSE;
   M4_ND_KK_1_1.CMD.Alarm := FALSE;
   M4_ND_KK_1_1.CMD.Reset := FALSE;
   M4_ND_KK_1_1.CMD.Sim := FALSE;
   M4_ND_KK_1_1.CMD.Vector := FALSE;
   M4_ND_KK_1_1.CMD.Ready := FALSE;
   M4_ND_KK_1_1.CMD.Resourse := FALSE;
   M4_ND_KK_1_1.T_ON := 0;
   M4_ND_KK_1_1.T_OFF := 0;
   M4_ND_KK_1_1.SP_M := 0.0;
   M4_ND_KK_1_1.Converter.Min_Out := 0.0;
   M4_ND_KK_1_1.Converter.Max_Out := 15.6;
   M5_ND_KK_1_2.CMD.Hand := FALSE;
   M5_ND_KK_1_2.CMD.Start_A := FALSE;
   M5_ND_KK_1_2.CMD.Start_M := FALSE;
   M5_ND_KK_1_2.CMD.Force := FALSE;
   M5_ND_KK_1_2.CMD.Lock := FALSE;
   M5_ND_KK_1_2.CMD.Local := FALSE;
   M5_ND_KK_1_2.CMD.Service := FALSE;
   M5_ND_KK_1_2.CMD.Safety := FALSE;
   M5_ND_KK_1_2.CMD.Alarm := FALSE;
   M5_ND_KK_1_2.CMD.Reset := FALSE;
   M5_ND_KK_1_2.CMD.Sim := FALSE;
   M5_ND_KK_1_2.CMD.Vector := FALSE;
   M5_ND_KK_1_2.CMD.Ready := FALSE;
   M5_ND_KK_1_2.CMD.Resourse := FALSE;
   M5_ND_KK_1_2.T_ON := 0;
   M5_ND_KK_1_2.T_OFF := 0;
   M5_ND_KK_1_2.SP_M := 0.0;
   M5_ND_KK_1_2.Converter.Min_Out := 0.0;
   M5_ND_KK_1_2.Converter.Max_Out := 15.6;
   M14_ND_K_1_1.CMD.Hand := FALSE;
   M14_ND_K_1_1.CMD.Start_A := FALSE;
   M14_ND_K_1_1.CMD.Start_M := FALSE;
   M14_ND_K_1_1.CMD.Force := FALSE;
   M14_ND_K_1_1.CMD.Lock := FALSE;
   M14_ND_K_1_1.CMD.Local := FALSE;
   M14_ND_K_1_1.CMD.Service := FALSE;
   M14_ND_K_1_1.CMD.Safety := FALSE;
   M14_ND_K_1_1.CMD.Alarm := FALSE;
   M14_ND_K_1_1.CMD.Reset := FALSE;
   M14_ND_K_1_1.CMD.Sim := FALSE;
   M14_ND_K_1_1.CMD.Vector := FALSE;
   M14_ND_K_1_1.CMD.Ready := FALSE;
   M14_ND_K_1_1.CMD.Resourse := FALSE;
   M14_ND_K_1_1.T_ON := 0;
   M14_ND_K_1_1.T_OFF := 0;
   M14_ND_K_1_1.SP_M := 0.0;
   M14_ND_K_1_1.Converter.Min_Out := 0.0;
   M14_ND_K_1_1.Converter.Max_Out := 15.6;
   M15_ND_K_1_2.CMD.Hand := FALSE;
   M15_ND_K_1_2.CMD.Start_A := FALSE;
   M15_ND_K_1_2.CMD.Start_M := FALSE;
   M15_ND_K_1_2.CMD.Force := FALSE;
   M15_ND_K_1_2.CMD.Lock := FALSE;
   M15_ND_K_1_2.CMD.Local := FALSE;
   M15_ND_K_1_2.CMD.Service := FALSE;
   M15_ND_K_1_2.CMD.Safety := FALSE;
   M15_ND_K_1_2.CMD.Alarm := FALSE;
   M15_ND_K_1_2.CMD.Reset := FALSE;
   M15_ND_K_1_2.CMD.Sim := FALSE;
   M15_ND_K_1_2.CMD.Vector := FALSE;
   M15_ND_K_1_2.CMD.Ready := FALSE;
   M15_ND_K_1_2.CMD.Resourse := FALSE;
   M15_ND_K_1_2.T_ON := 0;
   M15_ND_K_1_2.T_OFF := 0;
   M15_ND_K_1_2.SP_M := 0.0;
   M15_ND_K_1_2.Converter.Min_Out := 0.0;
   M15_ND_K_1_2.Converter.Max_Out := 15.6;
   M16_ND_K_1_3.CMD.Hand := FALSE;
   M16_ND_K_1_3.CMD.Start_A := FALSE;
   M16_ND_K_1_3.CMD.Start_M := FALSE;
   M16_ND_K_1_3.CMD.Force := FALSE;
   M16_ND_K_1_3.CMD.Lock := FALSE;
   M16_ND_K_1_3.CMD.Local := FALSE;
   M16_ND_K_1_3.CMD.Service := FALSE;
   M16_ND_K_1_3.CMD.Safety := FALSE;
   M16_ND_K_1_3.CMD.Alarm := FALSE;
   M16_ND_K_1_3.CMD.Reset := FALSE;
   M16_ND_K_1_3.CMD.Sim := FALSE;
   M16_ND_K_1_3.CMD.Vector := FALSE;
   M16_ND_K_1_3.CMD.Ready := FALSE;
   M16_ND_K_1_3.CMD.Resourse := FALSE;
   M16_ND_K_1_3.T_ON := 0;
   M16_ND_K_1_3.T_OFF := 0;
   M16_ND_K_1_3.SP_M := 0.0;
   M16_ND_K_1_3.Converter.Min_Out := 0.0;
   M16_ND_K_1_3.Converter.Max_Out := 15.6;
   M17_ND_K_2_1.CMD.Hand := FALSE;
   M17_ND_K_2_1.CMD.Start_A := FALSE;
   M17_ND_K_2_1.CMD.Start_M := FALSE;
   M17_ND_K_2_1.CMD.Force := FALSE;
   M17_ND_K_2_1.CMD.Lock := FALSE;
   M17_ND_K_2_1.CMD.Local := FALSE;
   M17_ND_K_2_1.CMD.Service := FALSE;
   M17_ND_K_2_1.CMD.Safety := FALSE;
   M17_ND_K_2_1.CMD.Alarm := FALSE;
   M17_ND_K_2_1.CMD.Reset := FALSE;
   M17_ND_K_2_1.CMD.Sim := FALSE;
   M17_ND_K_2_1.CMD.Vector := FALSE;
   M17_ND_K_2_1.CMD.Ready := FALSE;
   M17_ND_K_2_1.CMD.Resourse := FALSE;
   M17_ND_K_2_1.T_ON := 0;
   M17_ND_K_2_1.T_OFF := 0;
   M17_ND_K_2_1.SP_M := 0.0;
   M17_ND_K_2_1.Converter.Min_Out := 0.0;
   M17_ND_K_2_1.Converter.Max_Out := 15.6;
   M18_ND_K_2_2.CMD.Hand := FALSE;
   M18_ND_K_2_2.CMD.Start_A := FALSE;
   M18_ND_K_2_2.CMD.Start_M := FALSE;
   M18_ND_K_2_2.CMD.Force := FALSE;
   M18_ND_K_2_2.CMD.Lock := FALSE;
   M18_ND_K_2_2.CMD.Local := FALSE;
   M18_ND_K_2_2.CMD.Service := FALSE;
   M18_ND_K_2_2.CMD.Safety := FALSE;
   M18_ND_K_2_2.CMD.Alarm := FALSE;
   M18_ND_K_2_2.CMD.Reset := FALSE;
   M18_ND_K_2_2.CMD.Sim := FALSE;
   M18_ND_K_2_2.CMD.Vector := FALSE;
   M18_ND_K_2_2.CMD.Ready := FALSE;
   M18_ND_K_2_2.CMD.Resourse := FALSE;
   M18_ND_K_2_2.T_ON := 0;
   M18_ND_K_2_2.T_OFF := 0;
   M18_ND_K_2_2.SP_M := 0.0;
   M18_ND_K_2_2.Converter.Min_Out := 0.0;
   M18_ND_K_2_2.Converter.Max_Out := 15.6;
   M19_ND_K_2_3.CMD.Hand := FALSE;
   M19_ND_K_2_3.CMD.Start_A := FALSE;
   M19_ND_K_2_3.CMD.Start_M := FALSE;
   M19_ND_K_2_3.CMD.Force := FALSE;
   M19_ND_K_2_3.CMD.Lock := FALSE;
   M19_ND_K_2_3.CMD.Local := FALSE;
   M19_ND_K_2_3.CMD.Service := FALSE;
   M19_ND_K_2_3.CMD.Safety := FALSE;
   M19_ND_K_2_3.CMD.Alarm := FALSE;
   M19_ND_K_2_3.CMD.Reset := FALSE;
   M19_ND_K_2_3.CMD.Sim := FALSE;
   M19_ND_K_2_3.CMD.Vector := FALSE;
   M19_ND_K_2_3.CMD.Ready := FALSE;
   M19_ND_K_2_3.CMD.Resourse := FALSE;
   M19_ND_K_2_3.T_ON := 0;
   M19_ND_K_2_3.T_OFF := 0;
   M19_ND_K_2_3.SP_M := 0.0;
   M19_ND_K_2_3.Converter.Min_Out := 0.0;
   M19_ND_K_2_3.Converter.Max_Out := 15.6;
   XVS_035.CMD.Hand := FALSE;
   XVS_035.CMD.Start_A := TRUE;
   XVS_035.CMD.Start_M := TRUE;
   XVS_035.CMD.Force := FALSE;
   XVS_035.CMD.Lock := FALSE;
   XVS_035.CMD.Local := FALSE;
   XVS_035.CMD.Service := FALSE;
   XVS_035.CMD.Safety := FALSE;
   XVS_035.CMD.Alarm := FALSE;
   XVS_035.CMD.Reset := FALSE;
   XVS_035.CMD.Sim := FALSE;
   XVS_035.CMD.Vector := FALSE;
   XVS_035.CMD.Ready := FALSE;
   XVS_035.CMD.Resourse := FALSE;
   XVS_036.CMD.Hand := FALSE;
   XVS_036.CMD.Start_A := TRUE;
   XVS_036.CMD.Start_M := TRUE;
   XVS_036.CMD.Force := FALSE;
   XVS_036.CMD.Lock := FALSE;
   XVS_036.CMD.Local := FALSE;
   XVS_036.CMD.Service := FALSE;
   XVS_036.CMD.Safety := FALSE;
   XVS_036.CMD.Alarm := FALSE;
   XVS_036.CMD.Reset := FALSE;
   XVS_036.CMD.Sim := FALSE;
   XVS_036.CMD.Vector := FALSE;
   XVS_036.CMD.Ready := FALSE;
   XVS_036.CMD.Resourse := FALSE;
   Z_GVM_x.CMD.Hand := FALSE;
   Z_GVM_x.CMD.Start_A := FALSE;
   Z_GVM_x.CMD.Start_M := FALSE;
   Z_GVM_x.CMD.Force := FALSE;
   Z_GVM_x.CMD.Lock := FALSE;
   Z_GVM_x.CMD.Local := FALSE;
   Z_GVM_x.CMD.Service := FALSE;
   Z_GVM_x.CMD.Safety := FALSE;
   Z_GVM_x.CMD.Alarm := FALSE;
   Z_GVM_x.CMD.Reset := FALSE;
   Z_GVM_x.CMD.Sim := FALSE;
   Z_GVM_x.CMD.Vector := FALSE;
   Z_GVM_x.CMD.Ready := FALSE;
   Z_GVM_x.CMD.Resourse := FALSE;
   Z_GVM_x.T_ON := 0;
   Z_GVM_x.T_OFF := 0;
END_DATA_BLOCK

DATA_BLOCK "DB_OUT"   // DB102
{ S7_Optimized_Access := 'FALSE' }
VERSION : 0.1
// stored: AutoNumber false, DBAccessibleFromOPCUA true, IsOnlyStoredInLoadMemory false, IsWriteProtectedInAS false
   VAR
      AI_FT_007 { S7_SetPoint := 'True'} : "Out_AI";
      AI_FT_008 { S7_SetPoint := 'True'} : "Out_AI";
      AI_FT_009 { S7_SetPoint := 'True'} : "Out_AI";
      AI_FT_010 { S7_SetPoint := 'True'} : "Out_AI";
      AI_LT_014 { S7_SetPoint := 'True'} : "Out_AI";
      AI_LT_015 { S7_SetPoint := 'True'} : "Out_AI";
      AI_LT_016 { S7_SetPoint := 'True'} : "Out_AI";
      AI_LT_019 { S7_SetPoint := 'True'} : "Out_AI";
      AI_PT_001 { S7_SetPoint := 'True'} : "Out_AI";
      AI_PT_002 { S7_SetPoint := 'True'} : "Out_AI";
      AI_PT_003 { S7_SetPoint := 'True'} : "Out_AI";
      AI_PT_004 { S7_SetPoint := 'True'} : "Out_AI";
      AI_PT_005 { S7_SetPoint := 'True'} : "Out_AI";
      AI_PT_006 { S7_SetPoint := 'True'} : "Out_AI";
      Z_GVM_020 { S7_SetPoint := 'True'} : "Out_Z";
      Z_GVM_021 { S7_SetPoint := 'True'} : "Out_Z";
      Z_GVM_022 { S7_SetPoint := 'True'} : "Out_Z";
      Z_GCM_023 { S7_SetPoint := 'True'} : "Out_Z";
      Z_GCM_024 { S7_SetPoint := 'True'} : "Out_Z";
      Z_GCM_025 { S7_SetPoint := 'True'} : "Out_Z";
      XVS_026 { S7_SetPoint := 'True'} : "InOut_DO";
      XVS_027 { S7_SetPoint := 'True'} : "InOut_DO";
      XVS_028 { S7_SetPoint := 'True'} : "InOut_DO";
      XVS_029 { S7_SetPoint := 'True'} : "InOut_DO";
      XVS_030 { S7_SetPoint := 'True'} : "InOut_DO";
      XVS_031 { S7_SetPoint := 'True'} : "InOut_DO";
      XVS_032 { S7_SetPoint := 'True'} : "InOut_DO";
      XVS_033 { S7_SetPoint := 'True'} : "InOut_DO";
      XVS_034 { S7_SetPoint := 'True'} : "InOut_DO";
      M6_M_K_1_1 { S7_SetPoint := 'True'} : "Out_MD";
      M7_M_K_1_2 { S7_SetPoint := 'True'} : "Out_MD";
      M8_M_K_1_3 { S7_SetPoint := 'True'} : "Out_MD";
      M11_M_K_2_1 { S7_SetPoint := 'True'} : "Out_MD";
      M12_M_K_2_2 { S7_SetPoint := 'True'} : "Out_MD";
      M13_M_K_2_3 { S7_SetPoint := 'True'} : "Out_MD";
      M9_SD { S7_SetPoint := 'True'} : "Out_MDA";
      M10_Vibro { S7_SetPoint := 'True'} : "Out_MD";
      M1_BK_1 { S7_SetPoint := 'True'} : "Out_MDA";
      M2_KK_1_1 { S7_SetPoint := 'True'} : "Out_MDA";
      M3_KK_1_2 { S7_SetPoint := 'True'} : "Out_MDA";
      M4_ND_KK_1_1 { S7_SetPoint := 'True'} : "Out_MDA";
      M5_ND_KK_1_2 { S7_SetPoint := 'True'} : "Out_MDA";
      M14_ND_K_1_1 { S7_SetPoint := 'True'} : "Out_MDA";
      M15_ND_K_1_2 { S7_SetPoint := 'True'} : "Out_MDA";
      M16_ND_K_1_3 { S7_SetPoint := 'True'} : "Out_MDA";
      M17_ND_K_2_1 { S7_SetPoint := 'True'} : "Out_MDA";
      M18_ND_K_2_2 { S7_SetPoint := 'True'} : "Out_MDA";
      M19_ND_K_2_3 { S7_SetPoint := 'True'} : "Out_MDA";
      DIx : Struct
         LS_017 : Bool := FALSE;
         LS_018 : Bool := TRUE;
         FIS_011 : Bool := FALSE;
         FIS_012 : Bool := FALSE;
         FIS_013 : Bool := FALSE;
         ALS_1 : Bool := FALSE;
         ALS_2 : Bool := FALSE;
         LOCAL { S7_SetPoint := 'True'} : Bool := FALSE;
         All_Block : Bool := FALSE;
         Start_1 : Bool := FALSE;
         Start_2 : Bool := FALSE;
         Start_3 : Bool := FALSE;
         LS_019 : Bool := FALSE;
      END_STRUCT;
      PolyMix_1 : Struct
         Start : Bool := FALSE;
         SP_C : Real := 0.0;
         Messages : Struct
            Flow_Dry_Run : Bool := FALSE;
            Flow_Low : Bool := FALSE;
            LE_NoChange : Bool := FALSE;
            LE_Low : Bool := FALSE;
            LE_High : Bool := FALSE;
            LS_Low : Bool := FALSE;
            LS_NoProduct : Bool := FALSE;
            LS_Filter : Bool := FALSE;
            SD_Low : Bool := FALSE;
            Low_Weight : Bool := FALSE;
            Link_Error : Bool := FALSE;
            Alarm : Word := 16#0000;
         END_STRUCT;
      END_STRUCT;
      PolyMix_2 : Struct
         Start : Bool := FALSE;
         SP_C : Real := 0.0;
         Messages : Struct
            Flow_Dry_Run : Bool := FALSE;
            Flow_Low : Bool := FALSE;
            LE_NoChange : Bool := FALSE;
            LE_Low : Bool := FALSE;
            LE_High : Bool := FALSE;
            LS_Low : Bool := FALSE;
            LS_NoProduct : Bool := FALSE;
            LS_Filter : Bool := FALSE;
            SD_Low : Bool := FALSE;
            Low_Weight : Bool := FALSE;
            Link_Error : Bool := FALSE;
            Alarm : Word := 16#0000;
         END_STRUCT;
      END_STRUCT;
      XVS_035 { S7_SetPoint := 'True'} : "InOut_DO";
      XVS_036 { S7_SetPoint := 'True'} : "InOut_DO";
      gsm3_PolyMix_1 { S7_SetPoint := 'True'} : Real := 1.09;
      gsm3_PolyMix_2 : Real := 1.072;
      F1_Clean_Now : Bool := FALSE;
      F2_Clean_Now : Bool := FALSE;
      ALARM_NO_AIR : Bool := FALSE;
      Z_GVM_x { S7_SetPoint := 'True'} : "Out_Z";
      M_Vent : "Out_MD";
      Any_Alarms : Word := 16#0000;
      Events : Word := 16#0000;
      Lines : Array[1..7] of Struct
         Alarms : Word;
      END_STRUCT;
      res_5 : Word := 16#0000;
      res_6 : Word := 16#0000;
      res_7 : Word := 16#0000;
      res_8 : Word := 16#0000;
      res_9 : Word := 16#0000;
      res_10 : Word := 16#0000;
      Time_DTL { S7_SetPoint := 'True'} : DTL := DTL#2020-06-25-13:08:09.170187013;
   END_VAR
BEGIN
   AI_FT_007.Result := 0.04701968;
   AI_FT_007.Converter.Min_Out := 0.0;
   AI_FT_007.Converter.Max_Out := 1000.0;
   AI_FT_007.Alarms := 16#0000;
   AI_FT_007.SP.HH := 320.0;
   AI_FT_007.SP.H := 300.0;
   AI_FT_007.SP.L := 200.0;
   AI_FT_007.SP.LL := 75.0;
   AI_FT_008.Result := 0.02821181;
   AI_FT_008.Converter.Min_Out := 0.0;
   AI_FT_008.Converter.Max_Out := 100.0;
   AI_FT_008.Alarms := 16#0000;
   AI_FT_008.SP.HH := 100.0;
   AI_FT_008.SP.H := 15.0;
   AI_FT_008.SP.L := 0.5;
   AI_FT_008.SP.LL := -0.1;
   AI_FT_009.Result := 0.003616898;
   AI_FT_009.Converter.Min_Out := 0.0;
   AI_FT_009.Converter.Max_Out := 100.0;
   AI_FT_009.Alarms := 16#0000;
   AI_FT_009.SP.HH := 30.0;
   AI_FT_009.SP.H := 15.0;
   AI_FT_009.SP.L := 0.5;
   AI_FT_009.SP.LL := -0.1;
   AI_FT_010.Result := 0.01989294;
   AI_FT_010.Converter.Min_Out := 0.0;
   AI_FT_010.Converter.Max_Out := 100.0;
   AI_FT_010.Alarms := 16#0000;
   AI_FT_010.SP.HH := 50.0;
   AI_FT_010.SP.H := 40.0;
   AI_FT_010.SP.L := 0.5;
   AI_FT_010.SP.LL := -0.5;
   AI_LT_014.Result := 953.6309;
   AI_LT_014.Converter.Min_Out := 0.0;
   AI_LT_014.Converter.Max_Out := 2605.0;
   AI_LT_014.Alarms := 16#0000;
   AI_LT_014.SP.HH := 2400.0;
   AI_LT_014.SP.H := 2300.0;
   AI_LT_014.SP.L := 400.0;
   AI_LT_014.SP.LL := 220.0;
   AI_LT_015.Result := 2297.691;
   AI_LT_015.Converter.Min_Out := 0.0;
   AI_LT_015.Converter.Max_Out := 2605.0;
   AI_LT_015.Alarms := 16#0000;
   AI_LT_015.SP.HH := 2400.0;
   AI_LT_015.SP.H := 2300.0;
   AI_LT_015.SP.L := 400.0;
   AI_LT_015.SP.LL := 220.0;
   AI_LT_016.Result := 985.5756;
   AI_LT_016.Converter.Min_Out := 0.0;
   AI_LT_016.Converter.Max_Out := 1268.0;
   AI_LT_016.Alarms := 16#0004;
   AI_LT_016.SP.HH := 1060.0;
   AI_LT_016.SP.H := 950.0;
   AI_LT_016.SP.L := 250.0;
   AI_LT_016.SP.LL := 120.0;
   AI_LT_019.Result := 916.5906;
   AI_LT_019.Converter.Min_Out := 0.0;
   AI_LT_019.Converter.Max_Out := 1268.0;
   AI_LT_019.Alarms := 16#0000;
   AI_LT_019.SP.HH := 1060.0;
   AI_LT_019.SP.H := 950.0;
   AI_LT_019.SP.L := 250.0;
   AI_LT_019.SP.LL := 120.0;
   AI_PT_001.Result := 0.02823567;
   AI_PT_001.Converter.Min_Out := 0.0;
   AI_PT_001.Converter.Max_Out := 0.6;
   AI_PT_001.Alarms := 16#0000;
   AI_PT_001.SP.HH := 0.35;
   AI_PT_001.SP.H := 0.3;
   AI_PT_001.SP.L := 0.02;
   AI_PT_001.SP.LL := 0.01;
   AI_PT_002.Result := 0.02846354;
   AI_PT_002.Converter.Min_Out := 0.0;
   AI_PT_002.Converter.Max_Out := 0.6;
   AI_PT_002.Alarms := 16#0000;
   AI_PT_002.SP.HH := 0.35;
   AI_PT_002.SP.H := 0.3;
   AI_PT_002.SP.L := 0.02;
   AI_PT_002.SP.LL := 0.01;
   AI_PT_003.Result := 0.02719184;
   AI_PT_003.Converter.Min_Out := 0.0;
   AI_PT_003.Converter.Max_Out := 0.6;
   AI_PT_003.Alarms := 16#0000;
   AI_PT_003.SP.HH := 0.35;
   AI_PT_003.SP.H := 0.3;
   AI_PT_003.SP.L := 0.02;
   AI_PT_003.SP.LL := 0.01;
   AI_PT_004.Result := 0.02914063;
   AI_PT_004.Converter.Min_Out := 0.0;
   AI_PT_004.Converter.Max_Out := 0.6;
   AI_PT_004.Alarms := 16#0000;
   AI_PT_004.SP.HH := 0.35;
   AI_PT_004.SP.H := 0.3;
   AI_PT_004.SP.L := 0.02;
   AI_PT_004.SP.LL := 0.01;
   AI_PT_005.Result := 0.02641927;
   AI_PT_005.Converter.Min_Out := 0.0;
   AI_PT_005.Converter.Max_Out := 0.6;
   AI_PT_005.Alarms := 16#0000;
   AI_PT_005.SP.HH := 0.35;
   AI_PT_005.SP.H := 0.3;
   AI_PT_005.SP.L := 0.02;
   AI_PT_005.SP.LL := 0.01;
   AI_PT_006.Result := 0.02695746;
   AI_PT_006.Converter.Min_Out := 0.0;
   AI_PT_006.Converter.Max_Out := 0.6;
   AI_PT_006.Alarms := 16#0000;
   AI_PT_006.SP.HH := 0.35;
   AI_PT_006.SP.H := 0.3;
   AI_PT_006.SP.L := 0.02;
   AI_PT_006.SP.LL := 0.01;
   Z_GVM_020.CMD.Hand := FALSE;
   Z_GVM_020.CMD.Start_A := FALSE;
   Z_GVM_020.CMD.Start_M := FALSE;
   Z_GVM_020.CMD.Force := FALSE;
   Z_GVM_020.CMD.Lock := FALSE;
   Z_GVM_020.CMD.Local := FALSE;
   Z_GVM_020.CMD.Service := FALSE;
   Z_GVM_020.CMD.Safety := FALSE;
   Z_GVM_020.CMD.Alarm := FALSE;
   Z_GVM_020.CMD.Reset := FALSE;
   Z_GVM_020.CMD.Sim := FALSE;
   Z_GVM_020.CMD.Vector := FALSE;
   Z_GVM_020.CMD.Ready := FALSE;
   Z_GVM_020.CMD.Resourse := FALSE;
   Z_GVM_020.Status := 0;
   Z_GVM_020.T_ON := 12;
   Z_GVM_020.T_OFF := 12;
   Z_GVM_020.Alarms := 16#0000;
   Z_GVM_021.CMD.Hand := FALSE;
   Z_GVM_021.CMD.Start_A := FALSE;
   Z_GVM_021.CMD.Start_M := FALSE;
   Z_GVM_021.CMD.Force := FALSE;
   Z_GVM_021.CMD.Lock := FALSE;
   Z_GVM_021.CMD.Local := FALSE;
   Z_GVM_021.CMD.Service := FALSE;
   Z_GVM_021.CMD.Safety := FALSE;
   Z_GVM_021.CMD.Alarm := FALSE;
   Z_GVM_021.CMD.Reset := FALSE;
   Z_GVM_021.CMD.Sim := FALSE;
   Z_GVM_021.CMD.Vector := FALSE;
   Z_GVM_021.CMD.Ready := FALSE;
   Z_GVM_021.CMD.Resourse := FALSE;
   Z_GVM_021.Status := 0;
   Z_GVM_021.T_ON := 12;
   Z_GVM_021.T_OFF := 12;
   Z_GVM_021.Alarms := 16#0000;
   Z_GVM_022.CMD.Hand := FALSE;
   Z_GVM_022.CMD.Start_A := FALSE;
   Z_GVM_022.CMD.Start_M := FALSE;
   Z_GVM_022.CMD.Force := FALSE;
   Z_GVM_022.CMD.Lock := FALSE;
   Z_GVM_022.CMD.Local := FALSE;
   Z_GVM_022.CMD.Service := FALSE;
   Z_GVM_022.CMD.Safety := FALSE;
   Z_GVM_022.CMD.Alarm := FALSE;
   Z_GVM_022.CMD.Reset := FALSE;
   Z_GVM_022.CMD.Sim := FALSE;
   Z_GVM_022.CMD.Vector := FALSE;
   Z_GVM_022.CMD.Ready := FALSE;
   Z_GVM_022.CMD.Resourse := FALSE;
   Z_GVM_022.Status := 0;
   Z_GVM_022.T_ON := 12;
   Z_GVM_022.T_OFF := 12;
   Z_GVM_022.Alarms := 16#0000;
   Z_GCM_023.CMD.Hand := FALSE;
   Z_GCM_023.CMD.Start_A := FALSE;
   Z_GCM_023.CMD.Start_M := FALSE;
   Z_GCM_023.CMD.Force := FALSE;
   Z_GCM_023.CMD.Lock := FALSE;
   Z_GCM_023.CMD.Local := FALSE;
   Z_GCM_023.CMD.Service := FALSE;
   Z_GCM_023.CMD.Safety := FALSE;
   Z_GCM_023.CMD.Alarm := FALSE;
   Z_GCM_023.CMD.Reset := FALSE;
   Z_GCM_023.CMD.Sim := FALSE;
   Z_GCM_023.CMD.Vector := FALSE;
   Z_GCM_023.CMD.Ready := FALSE;
   Z_GCM_023.CMD.Resourse := FALSE;
   Z_GCM_023.Status := 0;
   Z_GCM_023.T_ON := 12;
   Z_GCM_023.T_OFF := 12;
   Z_GCM_023.Alarms := 16#0000;
   Z_GCM_024.CMD.Hand := FALSE;
   Z_GCM_024.CMD.Start_A := FALSE;
   Z_GCM_024.CMD.Start_M := FALSE;
   Z_GCM_024.CMD.Force := FALSE;
   Z_GCM_024.CMD.Lock := FALSE;
   Z_GCM_024.CMD.Local := FALSE;
   Z_GCM_024.CMD.Service := FALSE;
   Z_GCM_024.CMD.Safety := FALSE;
   Z_GCM_024.CMD.Alarm := FALSE;
   Z_GCM_024.CMD.Reset := FALSE;
   Z_GCM_024.CMD.Sim := FALSE;
   Z_GCM_024.CMD.Vector := FALSE;
   Z_GCM_024.CMD.Ready := FALSE;
   Z_GCM_024.CMD.Resourse := FALSE;
   Z_GCM_024.Status := 0;
   Z_GCM_024.T_ON := 12;
   Z_GCM_024.T_OFF := 12;
   Z_GCM_024.Alarms := 16#0000;
   Z_GCM_025.CMD.Hand := FALSE;
   Z_GCM_025.CMD.Start_A := FALSE;
   Z_GCM_025.CMD.Start_M := FALSE;
   Z_GCM_025.CMD.Force := FALSE;
   Z_GCM_025.CMD.Lock := FALSE;
   Z_GCM_025.CMD.Local := FALSE;
   Z_GCM_025.CMD.Service := FALSE;
   Z_GCM_025.CMD.Safety := FALSE;
   Z_GCM_025.CMD.Alarm := FALSE;
   Z_GCM_025.CMD.Reset := FALSE;
   Z_GCM_025.CMD.Sim := FALSE;
   Z_GCM_025.CMD.Vector := FALSE;
   Z_GCM_025.CMD.Ready := FALSE;
   Z_GCM_025.CMD.Resourse := FALSE;
   Z_GCM_025.Status := 0;
   Z_GCM_025.T_ON := 12;
   Z_GCM_025.T_OFF := 12;
   Z_GCM_025.Alarms := 16#0000;
   XVS_026.CMD.Hand := FALSE;
   XVS_026.CMD.Start_A := FALSE;
   XVS_026.CMD.Start_M := FALSE;
   XVS_026.CMD.Force := FALSE;
   XVS_026.CMD.Lock := FALSE;
   XVS_026.CMD.Local := FALSE;
   XVS_026.CMD.Service := FALSE;
   XVS_026.CMD.Safety := FALSE;
   XVS_026.CMD.Alarm := FALSE;
   XVS_026.CMD.Reset := FALSE;
   XVS_026.CMD.Sim := FALSE;
   XVS_026.CMD.Vector := FALSE;
   XVS_026.CMD.Ready := FALSE;
   XVS_026.CMD.Resourse := FALSE;
   XVS_027.CMD.Hand := FALSE;
   XVS_027.CMD.Start_A := FALSE;
   XVS_027.CMD.Start_M := FALSE;
   XVS_027.CMD.Force := FALSE;
   XVS_027.CMD.Lock := FALSE;
   XVS_027.CMD.Local := FALSE;
   XVS_027.CMD.Service := FALSE;
   XVS_027.CMD.Safety := FALSE;
   XVS_027.CMD.Alarm := FALSE;
   XVS_027.CMD.Reset := FALSE;
   XVS_027.CMD.Sim := FALSE;
   XVS_027.CMD.Vector := FALSE;
   XVS_027.CMD.Ready := FALSE;
   XVS_027.CMD.Resourse := FALSE;
   XVS_028.CMD.Hand := FALSE;
   XVS_028.CMD.Start_A := FALSE;
   XVS_028.CMD.Start_M := FALSE;
   XVS_028.CMD.Force := FALSE;
   XVS_028.CMD.Lock := FALSE;
   XVS_028.CMD.Local := FALSE;
   XVS_028.CMD.Service := FALSE;
   XVS_028.CMD.Safety := FALSE;
   XVS_028.CMD.Alarm := FALSE;
   XVS_028.CMD.Reset := FALSE;
   XVS_028.CMD.Sim := FALSE;
   XVS_028.CMD.Vector := FALSE;
   XVS_028.CMD.Ready := FALSE;
   XVS_028.CMD.Resourse := FALSE;
   XVS_029.CMD.Hand := FALSE;
   XVS_029.CMD.Start_A := FALSE;
   XVS_029.CMD.Start_M := FALSE;
   XVS_029.CMD.Force := FALSE;
   XVS_029.CMD.Lock := FALSE;
   XVS_029.CMD.Local := FALSE;
   XVS_029.CMD.Service := FALSE;
   XVS_029.CMD.Safety := FALSE;
   XVS_029.CMD.Alarm := FALSE;
   XVS_029.CMD.Reset := FALSE;
   XVS_029.CMD.Sim := FALSE;
   XVS_029.CMD.Vector := FALSE;
   XVS_029.CMD.Ready := FALSE;
   XVS_029.CMD.Resourse := FALSE;
   XVS_030.CMD.Hand := FALSE;
   XVS_030.CMD.Start_A := FALSE;
   XVS_030.CMD.Start_M := FALSE;
   XVS_030.CMD.Force := FALSE;
   XVS_030.CMD.Lock := FALSE;
   XVS_030.CMD.Local := FALSE;
   XVS_030.CMD.Service := FALSE;
   XVS_030.CMD.Safety := FALSE;
   XVS_030.CMD.Alarm := FALSE;
   XVS_030.CMD.Reset := FALSE;
   XVS_030.CMD.Sim := FALSE;
   XVS_030.CMD.Vector := FALSE;
   XVS_030.CMD.Ready := FALSE;
   XVS_030.CMD.Resourse := FALSE;
   XVS_031.CMD.Hand := FALSE;
   XVS_031.CMD.Start_A := FALSE;
   XVS_031.CMD.Start_M := FALSE;
   XVS_031.CMD.Force := FALSE;
   XVS_031.CMD.Lock := FALSE;
   XVS_031.CMD.Local := FALSE;
   XVS_031.CMD.Service := FALSE;
   XVS_031.CMD.Safety := FALSE;
   XVS_031.CMD.Alarm := FALSE;
   XVS_031.CMD.Reset := FALSE;
   XVS_031.CMD.Sim := FALSE;
   XVS_031.CMD.Vector := FALSE;
   XVS_031.CMD.Ready := FALSE;
   XVS_031.CMD.Resourse := FALSE;
   XVS_032.CMD.Hand := FALSE;
   XVS_032.CMD.Start_A := FALSE;
   XVS_032.CMD.Start_M := FALSE;
   XVS_032.CMD.Force := FALSE;
   XVS_032.CMD.Lock := FALSE;
   XVS_032.CMD.Local := FALSE;
   XVS_032.CMD.Service := FALSE;
   XVS_032.CMD.Safety := FALSE;
   XVS_032.CMD.Alarm := FALSE;
   XVS_032.CMD.Reset := FALSE;
   XVS_032.CMD.Sim := FALSE;
   XVS_032.CMD.Vector := FALSE;
   XVS_032.CMD.Ready := FALSE;
   XVS_032.CMD.Resourse := FALSE;
   XVS_033.CMD.Hand := FALSE;
   XVS_033.CMD.Start_A := FALSE;
   XVS_033.CMD.Start_M := FALSE;
   XVS_033.CMD.Force := FALSE;
   XVS_033.CMD.Lock := FALSE;
   XVS_033.CMD.Local := FALSE;
   XVS_033.CMD.Service := FALSE;
   XVS_033.CMD.Safety := FALSE;
   XVS_033.CMD.Alarm := FALSE;
   XVS_033.CMD.Reset := FALSE;
   XVS_033.CMD.Sim := FALSE;
   XVS_033.CMD.Vector := FALSE;
   XVS_033.CMD.Ready := FALSE;
   XVS_033.CMD.Resourse := FALSE;
   XVS_034.CMD.Hand := FALSE;
   XVS_034.CMD.Start_A := FALSE;
   XVS_034.CMD.Start_M := FALSE;
   XVS_034.CMD.Force := FALSE;
   XVS_034.CMD.Lock := FALSE;
   XVS_034.CMD.Local := FALSE;
   XVS_034.CMD.Service := FALSE;
   XVS_034.CMD.Safety := FALSE;
   XVS_034.CMD.Alarm := FALSE;
   XVS_034.CMD.Reset := FALSE;
   XVS_034.CMD.Sim := FALSE;
   XVS_034.CMD.Vector := FALSE;
   XVS_034.CMD.Ready := FALSE;
   XVS_034.CMD.Resourse := FALSE;
   M6_M_K_1_1.CMD.Hand := FALSE;
   M6_M_K_1_1.CMD.Start_A := TRUE;
   M6_M_K_1_1.CMD.Start_M := TRUE;
   M6_M_K_1_1.CMD.Force := FALSE;
   M6_M_K_1_1.CMD.Lock := FALSE;
   M6_M_K_1_1.CMD.Local := FALSE;
   M6_M_K_1_1.CMD.Service := FALSE;
   M6_M_K_1_1.CMD.Safety := FALSE;
   M6_M_K_1_1.CMD.Alarm := FALSE;
   M6_M_K_1_1.CMD.Reset := FALSE;
   M6_M_K_1_1.CMD.Sim := FALSE;
   M6_M_K_1_1.CMD.Vector := FALSE;
   M6_M_K_1_1.CMD.Ready := FALSE;
   M6_M_K_1_1.CMD.Resourse := FALSE;
   M6_M_K_1_1.Status := 1;
   M6_M_K_1_1.T_ON := 2;
   M6_M_K_1_1.T_OFF := 2;
   M6_M_K_1_1.Alarms := 16#0000;
   M6_M_K_1_1.Res_h := 271;
   M7_M_K_1_2.CMD.Hand := FALSE;
   M7_M_K_1_2.CMD.Start_A := TRUE;
   M7_M_K_1_2.CMD.Start_M := TRUE;
   M7_M_K_1_2.CMD.Force := FALSE;
   M7_M_K_1_2.CMD.Lock := FALSE;
   M7_M_K_1_2.CMD.Local := FALSE;
   M7_M_K_1_2.CMD.Service := FALSE;
   M7_M_K_1_2.CMD.Safety := FALSE;
   M7_M_K_1_2.CMD.Alarm := FALSE;
   M7_M_K_1_2.CMD.Reset := FALSE;
   M7_M_K_1_2.CMD.Sim := FALSE;
   M7_M_K_1_2.CMD.Vector := FALSE;
   M7_M_K_1_2.CMD.Ready := FALSE;
   M7_M_K_1_2.CMD.Resourse := FALSE;
   M7_M_K_1_2.Status := 1;
   M7_M_K_1_2.T_ON := 2;
   M7_M_K_1_2.T_OFF := 2;
   M7_M_K_1_2.Alarms := 16#0000;
   M7_M_K_1_2.Res_h := 133;
   M8_M_K_1_3.CMD.Hand := FALSE;
   M8_M_K_1_3.CMD.Start_A := TRUE;
   M8_M_K_1_3.CMD.Start_M := TRUE;
   M8_M_K_1_3.CMD.Force := FALSE;
   M8_M_K_1_3.CMD.Lock := FALSE;
   M8_M_K_1_3.CMD.Local := FALSE;
   M8_M_K_1_3.CMD.Service := FALSE;
   M8_M_K_1_3.CMD.Safety := FALSE;
   M8_M_K_1_3.CMD.Alarm := FALSE;
   M8_M_K_1_3.CMD.Reset := FALSE;
   M8_M_K_1_3.CMD.Sim := FALSE;
   M8_M_K_1_3.CMD.Vector := FALSE;
   M8_M_K_1_3.CMD.Ready := FALSE;
   M8_M_K_1_3.CMD.Resourse := FALSE;
   M8_M_K_1_3.Status := 1;
   M8_M_K_1_3.T_ON := 2;
   M8_M_K_1_3.T_OFF := 2;
   M8_M_K_1_3.Alarms := 16#0000;
   M8_M_K_1_3.Res_h := 269;
   M11_M_K_2_1.CMD.Hand := FALSE;
   M11_M_K_2_1.CMD.Start_A := FALSE;
   M11_M_K_2_1.CMD.Start_M := FALSE;
   M11_M_K_2_1.CMD.Force := FALSE;
   M11_M_K_2_1.CMD.Lock := FALSE;
   M11_M_K_2_1.CMD.Local := FALSE;
   M11_M_K_2_1.CMD.Service := FALSE;
   M11_M_K_2_1.CMD.Safety := FALSE;
   M11_M_K_2_1.CMD.Alarm := FALSE;
   M11_M_K_2_1.CMD.Reset := FALSE;
   M11_M_K_2_1.CMD.Sim := FALSE;
   M11_M_K_2_1.CMD.Vector := FALSE;
   M11_M_K_2_1.CMD.Ready := FALSE;
   M11_M_K_2_1.CMD.Resourse := FALSE;
   M11_M_K_2_1.Status := 0;
   M11_M_K_2_1.T_ON := 2;
   M11_M_K_2_1.T_OFF := 2;
   M11_M_K_2_1.Alarms := 16#0000;
   M11_M_K_2_1.Res_h := 227;
   M12_M_K_2_2.CMD.Hand := FALSE;
   M12_M_K_2_2.CMD.Start_A := FALSE;
   M12_M_K_2_2.CMD.Start_M := FALSE;
   M12_M_K_2_2.CMD.Force := FALSE;
   M12_M_K_2_2.CMD.Lock := FALSE;
   M12_M_K_2_2.CMD.Local := FALSE;
   M12_M_K_2_2.CMD.Service := FALSE;
   M12_M_K_2_2.CMD.Safety := FALSE;
   M12_M_K_2_2.CMD.Alarm := FALSE;
   M12_M_K_2_2.CMD.Reset := FALSE;
   M12_M_K_2_2.CMD.Sim := FALSE;
   M12_M_K_2_2.CMD.Vector := FALSE;
   M12_M_K_2_2.CMD.Ready := FALSE;
   M12_M_K_2_2.CMD.Resourse := FALSE;
   M12_M_K_2_2.Status := 0;
   M12_M_K_2_2.T_ON := 2;
   M12_M_K_2_2.T_OFF := 2;
   M12_M_K_2_2.Alarms := 16#0000;
   M12_M_K_2_2.Res_h := 182;
   M13_M_K_2_3.CMD.Hand := FALSE;
   M13_M_K_2_3.CMD.Start_A := FALSE;
   M13_M_K_2_3.CMD.Start_M := FALSE;
   M13_M_K_2_3.CMD.Force := FALSE;
   M13_M_K_2_3.CMD.Lock := FALSE;
   M13_M_K_2_3.CMD.Local := FALSE;
   M13_M_K_2_3.CMD.Service := FALSE;
   M13_M_K_2_3.CMD.Safety := FALSE;
   M13_M_K_2_3.CMD.Alarm := FALSE;
   M13_M_K_2_3.CMD.Reset := FALSE;
   M13_M_K_2_3.CMD.Sim := FALSE;
   M13_M_K_2_3.CMD.Vector := FALSE;
   M13_M_K_2_3.CMD.Ready := FALSE;
   M13_M_K_2_3.CMD.Resourse := FALSE;
   M13_M_K_2_3.Status := 0;
   M13_M_K_2_3.T_ON := 2;
   M13_M_K_2_3.T_OFF := 2;
   M13_M_K_2_3.Alarms := 16#0000;
   M13_M_K_2_3.Res_h := 163;
   M9_SD.CMD.Hand := FALSE;
   M9_SD.CMD.Start_A := FALSE;
   M9_SD.CMD.Start_M := FALSE;
   M9_SD.CMD.Force := FALSE;
   M9_SD.CMD.Lock := FALSE;
   M9_SD.CMD.Local := FALSE;
   M9_SD.CMD.Service := FALSE;
   M9_SD.CMD.Safety := FALSE;
   M9_SD.CMD.Alarm := FALSE;
   M9_SD.CMD.Reset := FALSE;
   M9_SD.CMD.Sim := FALSE;
   M9_SD.CMD.Vector := FALSE;
   M9_SD.CMD.Ready := FALSE;
   M9_SD.CMD.Resourse := FALSE;
   M9_SD.Status := 0;
   M9_SD.T_ON := 2;
   M9_SD.T_OFF := 2;
   M9_SD.Alarms := 16#0000;
   M9_SD.Res_h := 26;
   M9_SD.SP_M := 0.0;
   M9_SD.Converter.Min_Out := 0.0;
   M9_SD.Converter.Max_Out := 100.0;
   M10_Vibro.CMD.Hand := FALSE;
   M10_Vibro.CMD.Start_A := FALSE;
   M10_Vibro.CMD.Start_M := FALSE;
   M10_Vibro.CMD.Force := FALSE;
   M10_Vibro.CMD.Lock := FALSE;
   M10_Vibro.CMD.Local := FALSE;
   M10_Vibro.CMD.Service := FALSE;
   M10_Vibro.CMD.Safety := FALSE;
   M10_Vibro.CMD.Alarm := FALSE;
   M10_Vibro.CMD.Reset := FALSE;
   M10_Vibro.CMD.Sim := FALSE;
   M10_Vibro.CMD.Vector := FALSE;
   M10_Vibro.CMD.Ready := FALSE;
   M10_Vibro.CMD.Resourse := FALSE;
   M10_Vibro.Status := 0;
   M10_Vibro.T_ON := 2;
   M10_Vibro.T_OFF := 2;
   M10_Vibro.Alarms := 16#0000;
   M10_Vibro.Res_h := 0;
   M1_BK_1.CMD.Hand := FALSE;
   M1_BK_1.CMD.Start_A := FALSE;
   M1_BK_1.CMD.Start_M := FALSE;
   M1_BK_1.CMD.Force := FALSE;
   M1_BK_1.CMD.Lock := TRUE;
   M1_BK_1.CMD.Local := FALSE;
   M1_BK_1.CMD.Service := FALSE;
   M1_BK_1.CMD.Safety := FALSE;
   M1_BK_1.CMD.Alarm := FALSE;
   M1_BK_1.CMD.Reset := FALSE;
   M1_BK_1.CMD.Sim := FALSE;
   M1_BK_1.CMD.Vector := FALSE;
   M1_BK_1.CMD.Ready := FALSE;
   M1_BK_1.CMD.Resourse := FALSE;
   M1_BK_1.Status := 0;
   M1_BK_1.T_ON := 2;
   M1_BK_1.T_OFF := 2;
   M1_BK_1.Alarms := 16#0000;
   M1_BK_1.Res_h := 2;
   M1_BK_1.SP_M := 100.0;
   M1_BK_1.Converter.Min_Out := 0.0;
   M1_BK_1.Converter.Max_Out := 0.0;
   M2_KK_1_1.CMD.Hand := FALSE;
   M2_KK_1_1.CMD.Start_A := FALSE;
   M2_KK_1_1.CMD.Start_M := FALSE;
   M2_KK_1_1.CMD.Force := FALSE;
   M2_KK_1_1.CMD.Lock := TRUE;
   M2_KK_1_1.CMD.Local := FALSE;
   M2_KK_1_1.CMD.Service := FALSE;
   M2_KK_1_1.CMD.Safety := FALSE;
   M2_KK_1_1.CMD.Alarm := FALSE;
   M2_KK_1_1.CMD.Reset := FALSE;
   M2_KK_1_1.CMD.Sim := FALSE;
   M2_KK_1_1.CMD.Vector := FALSE;
   M2_KK_1_1.CMD.Ready := FALSE;
   M2_KK_1_1.CMD.Resourse := FALSE;
   M2_KK_1_1.Status := 0;
   M2_KK_1_1.T_ON := 2;
   M2_KK_1_1.T_OFF := 2;
   M2_KK_1_1.Alarms := 16#0000;
   M2_KK_1_1.Res_h := 2;
   M2_KK_1_1.SP_M := 0.0;
   M2_KK_1_1.Converter.Min_Out := 0.0;
   M2_KK_1_1.Converter.Max_Out := 0.0;
   M3_KK_1_2.CMD.Hand := FALSE;
   M3_KK_1_2.CMD.Start_A := FALSE;
   M3_KK_1_2.CMD.Start_M := FALSE;
   M3_KK_1_2.CMD.Force := FALSE;
   M3_KK_1_2.CMD.Lock := TRUE;
   M3_KK_1_2.CMD.Local := FALSE;
   M3_KK_1_2.CMD.Service := FALSE;
   M3_KK_1_2.CMD.Safety := FALSE;
   M3_KK_1_2.CMD.Alarm := FALSE;
   M3_KK_1_2.CMD.Reset := FALSE;
   M3_KK_1_2.CMD.Sim := FALSE;
   M3_KK_1_2.CMD.Vector := FALSE;
   M3_KK_1_2.CMD.Ready := FALSE;
   M3_KK_1_2.CMD.Resourse := FALSE;
   M3_KK_1_2.Status := 0;
   M3_KK_1_2.T_ON := 2;
   M3_KK_1_2.T_OFF := 2;
   M3_KK_1_2.Alarms := 16#0000;
   M3_KK_1_2.Res_h := 0;
   M3_KK_1_2.SP_M := 0.0;
   M3_KK_1_2.Converter.Min_Out := 0.0;
   M3_KK_1_2.Converter.Max_Out := 0.0;
   M4_ND_KK_1_1.CMD.Hand := FALSE;
   M4_ND_KK_1_1.CMD.Start_A := FALSE;
   M4_ND_KK_1_1.CMD.Start_M := FALSE;
   M4_ND_KK_1_1.CMD.Force := FALSE;
   M4_ND_KK_1_1.CMD.Lock := TRUE;
   M4_ND_KK_1_1.CMD.Local := FALSE;
   M4_ND_KK_1_1.CMD.Service := FALSE;
   M4_ND_KK_1_1.CMD.Safety := FALSE;
   M4_ND_KK_1_1.CMD.Alarm := FALSE;
   M4_ND_KK_1_1.CMD.Reset := FALSE;
   M4_ND_KK_1_1.CMD.Sim := FALSE;
   M4_ND_KK_1_1.CMD.Vector := FALSE;
   M4_ND_KK_1_1.CMD.Ready := FALSE;
   M4_ND_KK_1_1.CMD.Resourse := FALSE;
   M4_ND_KK_1_1.Status := 0;
   M4_ND_KK_1_1.T_ON := 0;
   M4_ND_KK_1_1.T_OFF := 0;
   M4_ND_KK_1_1.Alarms := 16#0000;
   M4_ND_KK_1_1.Res_h := 1;
   M4_ND_KK_1_1.SP_M := 0.0;
   M4_ND_KK_1_1.Converter.Min_Out := 0.0;
   M4_ND_KK_1_1.Converter.Max_Out := 15.6;
   M5_ND_KK_1_2.CMD.Hand := FALSE;
   M5_ND_KK_1_2.CMD.Start_A := FALSE;
   M5_ND_KK_1_2.CMD.Start_M := FALSE;
   M5_ND_KK_1_2.CMD.Force := FALSE;
   M5_ND_KK_1_2.CMD.Lock := TRUE;
   M5_ND_KK_1_2.CMD.Local := FALSE;
   M5_ND_KK_1_2.CMD.Service := FALSE;
   M5_ND_KK_1_2.CMD.Safety := FALSE;
   M5_ND_KK_1_2.CMD.Alarm := FALSE;
   M5_ND_KK_1_2.CMD.Reset := FALSE;
   M5_ND_KK_1_2.CMD.Sim := FALSE;
   M5_ND_KK_1_2.CMD.Vector := FALSE;
   M5_ND_KK_1_2.CMD.Ready := FALSE;
   M5_ND_KK_1_2.CMD.Resourse := FALSE;
   M5_ND_KK_1_2.Status := 0;
   M5_ND_KK_1_2.T_ON := 0;
   M5_ND_KK_1_2.T_OFF := 0;
   M5_ND_KK_1_2.Alarms := 16#0000;
   M5_ND_KK_1_2.Res_h := 5;
   M5_ND_KK_1_2.SP_M := 0.0;
   M5_ND_KK_1_2.Converter.Min_Out := 0.0;
   M5_ND_KK_1_2.Converter.Max_Out := 15.6;
   M14_ND_K_1_1.CMD.Hand := FALSE;
   M14_ND_K_1_1.CMD.Start_A := FALSE;
   M14_ND_K_1_1.CMD.Start_M := FALSE;
   M14_ND_K_1_1.CMD.Force := FALSE;
   M14_ND_K_1_1.CMD.Lock := FALSE;
   M14_ND_K_1_1.CMD.Local := FALSE;
   M14_ND_K_1_1.CMD.Service := FALSE;
   M14_ND_K_1_1.CMD.Safety := FALSE;
   M14_ND_K_1_1.CMD.Alarm := FALSE;
   M14_ND_K_1_1.CMD.Reset := FALSE;
   M14_ND_K_1_1.CMD.Sim := FALSE;
   M14_ND_K_1_1.CMD.Vector := FALSE;
   M14_ND_K_1_1.CMD.Ready := FALSE;
   M14_ND_K_1_1.CMD.Resourse := FALSE;
   M14_ND_K_1_1.Status := 0;
   M14_ND_K_1_1.T_ON := 0;
   M14_ND_K_1_1.T_OFF := 0;
   M14_ND_K_1_1.Alarms := 16#0000;
   M14_ND_K_1_1.Res_h := 42;
   M14_ND_K_1_1.SP_M := 0.0;
   M14_ND_K_1_1.Converter.Min_Out := 0.0;
   M14_ND_K_1_1.Converter.Max_Out := 15.6;
   M15_ND_K_1_2.CMD.Hand := FALSE;
   M15_ND_K_1_2.CMD.Start_A := FALSE;
   M15_ND_K_1_2.CMD.Start_M := FALSE;
   M15_ND_K_1_2.CMD.Force := FALSE;
   M15_ND_K_1_2.CMD.Lock := FALSE;
   M15_ND_K_1_2.CMD.Local := FALSE;
   M15_ND_K_1_2.CMD.Service := FALSE;
   M15_ND_K_1_2.CMD.Safety := FALSE;
   M15_ND_K_1_2.CMD.Alarm := FALSE;
   M15_ND_K_1_2.CMD.Reset := FALSE;
   M15_ND_K_1_2.CMD.Sim := FALSE;
   M15_ND_K_1_2.CMD.Vector := FALSE;
   M15_ND_K_1_2.CMD.Ready := FALSE;
   M15_ND_K_1_2.CMD.Resourse := FALSE;
   M15_ND_K_1_2.Status := 0;
   M15_ND_K_1_2.T_ON := 0;
   M15_ND_K_1_2.T_OFF := 0;
   M15_ND_K_1_2.Alarms := 16#0000;
   M15_ND_K_1_2.Res_h := 72;
   M15_ND_K_1_2.SP_M := 0.0;
   M15_ND_K_1_2.Converter.Min_Out := 0.0;
   M15_ND_K_1_2.Converter.Max_Out := 15.6;
   M16_ND_K_1_3.CMD.Hand := FALSE;
   M16_ND_K_1_3.CMD.Start_A := FALSE;
   M16_ND_K_1_3.CMD.Start_M := FALSE;
   M16_ND_K_1_3.CMD.Force := FALSE;
   M16_ND_K_1_3.CMD.Lock := FALSE;
   M16_ND_K_1_3.CMD.Local := FALSE;
   M16_ND_K_1_3.CMD.Service := FALSE;
   M16_ND_K_1_3.CMD.Safety := FALSE;
   M16_ND_K_1_3.CMD.Alarm := FALSE;
   M16_ND_K_1_3.CMD.Reset := FALSE;
   M16_ND_K_1_3.CMD.Sim := FALSE;
   M16_ND_K_1_3.CMD.Vector := FALSE;
   M16_ND_K_1_3.CMD.Ready := FALSE;
   M16_ND_K_1_3.CMD.Resourse := FALSE;
   M16_ND_K_1_3.Status := 0;
   M16_ND_K_1_3.T_ON := 0;
   M16_ND_K_1_3.T_OFF := 0;
   M16_ND_K_1_3.Alarms := 16#0000;
   M16_ND_K_1_3.Res_h := 11;
   M16_ND_K_1_3.SP_M := 0.0;
   M16_ND_K_1_3.Converter.Min_Out := 0.0;
   M16_ND_K_1_3.Converter.Max_Out := 15.6;
   M17_ND_K_2_1.CMD.Hand := FALSE;
   M17_ND_K_2_1.CMD.Start_A := FALSE;
   M17_ND_K_2_1.CMD.Start_M := FALSE;
   M17_ND_K_2_1.CMD.Force := FALSE;
   M17_ND_K_2_1.CMD.Lock := FALSE;
   M17_ND_K_2_1.CMD.Local := FALSE;
   M17_ND_K_2_1.CMD.Service := FALSE;
   M17_ND_K_2_1.CMD.Safety := FALSE;
   M17_ND_K_2_1.CMD.Alarm := FALSE;
   M17_ND_K_2_1.CMD.Reset := FALSE;
   M17_ND_K_2_1.CMD.Sim := FALSE;
   M17_ND_K_2_1.CMD.Vector := FALSE;
   M17_ND_K_2_1.CMD.Ready := FALSE;
   M17_ND_K_2_1.CMD.Resourse := FALSE;
   M17_ND_K_2_1.Status := 0;
   M17_ND_K_2_1.T_ON := 0;
   M17_ND_K_2_1.T_OFF := 0;
   M17_ND_K_2_1.Alarms := 16#0000;
   M17_ND_K_2_1.Res_h := 160;
   M17_ND_K_2_1.SP_M := 0.0;
   M17_ND_K_2_1.Converter.Min_Out := 0.0;
   M17_ND_K_2_1.Converter.Max_Out := 15.6;
   M18_ND_K_2_2.CMD.Hand := FALSE;
   M18_ND_K_2_2.CMD.Start_A := FALSE;
   M18_ND_K_2_2.CMD.Start_M := FALSE;
   M18_ND_K_2_2.CMD.Force := FALSE;
   M18_ND_K_2_2.CMD.Lock := FALSE;
   M18_ND_K_2_2.CMD.Local := FALSE;
   M18_ND_K_2_2.CMD.Service := FALSE;
   M18_ND_K_2_2.CMD.Safety := FALSE;
   M18_ND_K_2_2.CMD.Alarm := FALSE;
   M18_ND_K_2_2.CMD.Reset := FALSE;
   M18_ND_K_2_2.CMD.Sim := FALSE;
   M18_ND_K_2_2.CMD.Vector := FALSE;
   M18_ND_K_2_2.CMD.Ready := FALSE;
   M18_ND_K_2_2.CMD.Resourse := FALSE;
   M18_ND_K_2_2.Status := 0;
   M18_ND_K_2_2.T_ON := 0;
   M18_ND_K_2_2.T_OFF := 0;
   M18_ND_K_2_2.Alarms := 16#0000;
   M18_ND_K_2_2.Res_h := 1;
   M18_ND_K_2_2.SP_M := 0.0;
   M18_ND_K_2_2.Converter.Min_Out := 0.0;
   M18_ND_K_2_2.Converter.Max_Out := 15.6;
   M19_ND_K_2_3.CMD.Hand := FALSE;
   M19_ND_K_2_3.CMD.Start_A := FALSE;
   M19_ND_K_2_3.CMD.Start_M := FALSE;
   M19_ND_K_2_3.CMD.Force := FALSE;
   M19_ND_K_2_3.CMD.Lock := FALSE;
   M19_ND_K_2_3.CMD.Local := FALSE;
   M19_ND_K_2_3.CMD.Service := FALSE;
   M19_ND_K_2_3.CMD.Safety := FALSE;
   M19_ND_K_2_3.CMD.Alarm := FALSE;
   M19_ND_K_2_3.CMD.Reset := FALSE;
   M19_ND_K_2_3.CMD.Sim := FALSE;
   M19_ND_K_2_3.CMD.Vector := FALSE;
   M19_ND_K_2_3.CMD.Ready := FALSE;
   M19_ND_K_2_3.CMD.Resourse := FALSE;
   M19_ND_K_2_3.Status := 0;
   M19_ND_K_2_3.T_ON := 0;
   M19_ND_K_2_3.T_OFF := 0;
   M19_ND_K_2_3.Alarms := 16#0000;
   M19_ND_K_2_3.Res_h := 0;
   M19_ND_K_2_3.SP_M := 0.0;
   M19_ND_K_2_3.Converter.Min_Out := 0.0;
   M19_ND_K_2_3.Converter.Max_Out := 15.6;
   XVS_035.CMD.Hand := FALSE;
   XVS_035.CMD.Start_A := TRUE;
   XVS_035.CMD.Start_M := TRUE;
   XVS_035.CMD.Force := FALSE;
   XVS_035.CMD.Lock := FALSE;
   XVS_035.CMD.Local := FALSE;
   XVS_035.CMD.Service := FALSE;
   XVS_035.CMD.Safety := FALSE;
   XVS_035.CMD.Alarm := FALSE;
   XVS_035.CMD.Reset := FALSE;
   XVS_035.CMD.Sim := FALSE;
   XVS_035.CMD.Vector := FALSE;
   XVS_035.CMD.Ready := FALSE;
   XVS_035.CMD.Resourse := FALSE;
   XVS_036.CMD.Hand := FALSE;
   XVS_036.CMD.Start_A := TRUE;
   XVS_036.CMD.Start_M := TRUE;
   XVS_036.CMD.Force := FALSE;
   XVS_036.CMD.Lock := FALSE;
   XVS_036.CMD.Local := FALSE;
   XVS_036.CMD.Service := FALSE;
   XVS_036.CMD.Safety := FALSE;
   XVS_036.CMD.Alarm := FALSE;
   XVS_036.CMD.Reset := FALSE;
   XVS_036.CMD.Sim := FALSE;
   XVS_036.CMD.Vector := FALSE;
   XVS_036.CMD.Ready := FALSE;
   XVS_036.CMD.Resourse := FALSE;
   Z_GVM_x.CMD.Hand := FALSE;
   Z_GVM_x.CMD.Start_A := FALSE;
   Z_GVM_x.CMD.Start_M := FALSE;
   Z_GVM_x.CMD.Force := FALSE;
   Z_GVM_x.CMD.Lock := FALSE;
   Z_GVM_x.CMD.Local := FALSE;
   Z_GVM_x.CMD.Service := FALSE;
   Z_GVM_x.CMD.Safety := FALSE;
   Z_GVM_x.CMD.Alarm := FALSE;
   Z_GVM_x.CMD.Reset := FALSE;
   Z_GVM_x.CMD.Sim := FALSE;
   Z_GVM_x.CMD.Vector := FALSE;
   Z_GVM_x.CMD.Ready := FALSE;
   Z_GVM_x.CMD.Resourse := FALSE;
   Z_GVM_x.Status := 0;
   Z_GVM_x.T_ON := 0;
   Z_GVM_x.T_OFF := 0;
   Z_GVM_x.Alarms := 16#0000;
   M_Vent.CMD.Hand := FALSE;
   M_Vent.CMD.Start_A := FALSE;
   M_Vent.CMD.Start_M := FALSE;
   M_Vent.CMD.Force := FALSE;
   M_Vent.CMD.Lock := FALSE;
   M_Vent.CMD.Local := FALSE;
   M_Vent.CMD.Service := FALSE;
   M_Vent.CMD.Safety := FALSE;
   M_Vent.CMD.Alarm := FALSE;
   M_Vent.CMD.Reset := FALSE;
   M_Vent.CMD.Sim := FALSE;
   M_Vent.CMD.Vector := FALSE;
   M_Vent.CMD.Ready := FALSE;
   M_Vent.CMD.Resourse := FALSE;
   M_Vent.Status := 0;
   M_Vent.T_ON := 2;
   M_Vent.T_OFF := 2;
   M_Vent.Alarms := 16#0000;
   M_Vent.Res_h := 9;
   Lines[1..7].Alarms := 16#0000;
END_DATA_BLOCK

DATA_BLOCK "Report_Line_1_DB"   // DB51
{ S7_Optimized_Access := 'FALSE' }
VERSION : 0.1
// stored: AutoNumber false, DBAccessibleFromOPCUA true, IsOnlyStoredInLoadMemory false, IsWriteProtectedInAS false
   VAR RETAIN
      Report : Struct
         Last_Day : Int := 3;   // Прошедший день
         Last_Date : Int := 13;   // Прошедшее число (дата)
         Last_Month : Int := 10;   // Прошедший месяц
         RM_1 : Real := 0.0;   // Расходомер 1
         RM_2 : Real := 0.0;   // Расходомер 2
         D_Mid : Real := 0.0;   // Средняя доза за сутки
         Flow : Real := 0.0;   // Общая труба (куда происходит дозация)
         Days { S7_SetPoint := 'True'} : Array[1..7] of "Line_Report";   // Дни
         cnt : Int := 7;
         cnt_x : Int := 1;
      END_STRUCT;
      Report_H : "Line_Report";
      Time_DTL : DTL := DTL#2020-10-13-13:05:16.070116724;
   END_VAR
BEGIN
   Report.Days[1..2].RM_1 := 0.0;
   Report.Days[3].RM_1 := 870.1801;
   Report.Days[4].RM_1 := 870.2496;
   Report.Days[5].RM_1 := 991.9506;
   Report.Days[6].RM_1 := 829.0188;
   Report.Days[7].RM_1 := 13.7433;
   Report.Days[1..7].RM_2 := 0.0;
   Report.Days[1..7].Res_1 := 0.0;
   Report.Days[1..7].Res_2 := 0.0;
   Report.Days[1..2].D_Mid := 0.0;
   Report.Days[3].D_Mid := 3.5;
   Report.Days[4].D_Mid := 3.310966;
   Report.Days[5].D_Mid := 3.219339;
   Report.Days[6].D_Mid := 3.56408;
   Report.Days[7].D_Mid := 1.909127;
   Report.Days[1..2].Flow := 0.0;
   Report.Days[3].Flow := 13326.62;
   Report.Days[4].Flow := 14077.05;
   Report.Days[5].Flow := 16594.77;
   Report.Days[6].Flow := 12534.46;
   Report.Days[7].Flow := 344.1002;
   Report.Days[1].WeekDay := 2;
   Report.Days[2].WeekDay := 1;
   Report.Days[3].WeekDay := 7;
   Report.Days[4].WeekDay := 6;
   Report.Days[5].WeekDay := 5;
   Report.Days[6].WeekDay := 4;
   Report.Days[7].WeekDay := 3;
   Report.Days[1].Day := 12;
   Report.Days[2].Day := 11;
   Report.Days[3].Day := 10;
   Report.Days[4].Day := 9;
   Report.Days[5].Day := 8;
   Report.Days[6].Day := 7;
   Report.Days[7].Day := 6;
   Report.Days[1..7].Month := 10;
   Report_H.RM_1 := 0.0;
   Report_H.RM_2 := 0.0;
   Report_H.Res_1 := 9200.248;
   Report_H.Res_2 := 2713.0;
   Report_H.D_Mid := 3.391171;
   Report_H.Flow := 0.0;
   Report_H.WeekDay := 0;
   Report_H.Day := 0;
   Report_H.Month := 0;
END_DATA_BLOCK

DATA_BLOCK "Report_Line_2_DB"   // DB52
{ S7_Optimized_Access := 'FALSE' }
VERSION : 0.1
// stored: AutoNumber false, DBAccessibleFromOPCUA true, IsOnlyStoredInLoadMemory false, IsWriteProtectedInAS false
   VAR RETAIN
      Report : Struct
         Last_Day : Int := 3;   // Прошедший день
         Last_Date : Int := 13;   // Прошедшее число (дата)
         Last_Month : Int := 10;   // Прошедший месяц
         RM_1 : Real := 956.8786;   // Расходомер 1
         RM_2 : Real := 0.0;   // Расходомер 2
         D_Mid : Real := 3.0;   // Средняя доза за сутки
         Flow : Real := 17096.32;   // Общая труба (куда происходит дозация)
         Days { S7_SetPoint := 'True'} : Array[1..7] of "Line_Report";   // Дни
         cnt : Int := 7;
         cnt_x : Int := 1;
      END_STRUCT;
      Report_H : "Line_Report";
      Time_DTL : DTL := DTL#2020-10-13-13:05:16.588575848;
   END_VAR
BEGIN
   Report.Days[1].RM_1 := 1936.87;
   Report.Days[2].RM_1 := 2298.9;
   Report.Days[3].RM_1 := 1640.521;
   Report.Days[4].RM_1 := 43.10154;
   Report.Days[5].RM_1 := 5.310862;
   Report.Days[6].RM_1 := 0.0;
   Report.Days[7].RM_1 := 3.251781;
   Report.Days[1..7].RM_2 := 0.0;
   Report.Days[1..7].Res_1 := 0.0;
   Report.Days[1..7].Res_2 := 0.0;
   Report.Days[1].D_Mid := 3.046245;
   Report.Days[2..3].D_Mid := 3.5;
   Report.Days[4].D_Mid := 1.8125;
   Report.Days[5].D_Mid := 4.0;
   Report.Days[6].D_Mid := 0.0;
   Report.Days[7].D_Mid := 3.0;
   Report.Days[1].Flow := 34064.4;
   Report.Days[2].Flow := 35206.3;
   Report.Days[3].Flow := 25124.08;
   Report.Days[4].Flow := 1278.395;
   Report.Days[5].Flow := 77.60835;
   Report.Days[6].Flow := 0.0;
   Report.Days[7].Flow := 58.42366;
   Report.Days[1].WeekDay := 2;
   Report.Days[2].WeekDay := 1;
   Report.Days[3].WeekDay := 7;
   Report.Days[4].WeekDay := 6;
   Report.Days[5].WeekDay := 5;
   Report.Days[6].WeekDay := 4;
   Report.Days[7].WeekDay := 3;
   Report.Days[1].Day := 12;
   Report.Days[2].Day := 11;
   Report.Days[3].Day := 10;
   Report.Days[4].Day := 9;
   Report.Days[5].Day := 8;
   Report.Days[6].Day := 7;
   Report.Days[7].Day := 6;
   Report.Days[1..7].Month := 10;
   Report_H.RM_1 := 0.0;
   Report_H.RM_2 := 0.0;
   Report_H.Res_1 := 15224.0;
   Report_H.Res_2 := 4675.0;
   Report_H.D_Mid := 3.256471;
   Report_H.Flow := 0.0;
   Report_H.WeekDay := 0;
   Report_H.Day := 0;
   Report_H.Month := 0;
END_DATA_BLOCK

DATA_BLOCK "Support_DB"   // DB1000
{ S7_Optimized_Access := 'TRUE' }
VERSION : 0.1
// stored: AutoNumber false, DBAccessibleFromOPCUA true, IsOnlyStoredInLoadMemory false, IsRetainMemResEnabled false, IsWriteProtectedInAS false, MemoryReserve 100
   VAR
      DTR_Clean : Bool;   // Очистка DTR
      DTR_1 : Int;   // Data Transfer 1
      DTR_2 : Int;   // Data Transfer 2
      DTR_3 : Int;   // Data Transfer 3
   END_VAR
   VAR RETAIN
      All_AIs { S7_SetPoint := 'True'} : Int := 399;   // Номер последнего DB аналоговых входов
      All_AOs { S7_SetPoint := 'True'} : Int := 499;   // Номер последнего DB аналоговых выходов
      All_DIs { S7_SetPoint := 'True'} : Int := 209;   // Номер последнего DB дискретных входов
      All_DOs { S7_SetPoint := 'True'} : Int := 219;   // Номер последнего DB дискретных выходов
      All_MDs { S7_SetPoint := 'True'} : Int := 599;   // Номер последнего DB двигателей без ЧП
      All_MDAs { S7_SetPoint := 'True'} : Int := 699;   // Номер последнего DB двигателей с ЧП
      All_VD2s { S7_SetPoint := 'True'} : Int := 799;   // Номер последнего DB заслонки
      All_VD2As { S7_SetPoint := 'True'} : Int := 899;   // Номер последнего DB заслонки с позиционированием
      All_PIDs { S7_SetPoint := 'True'} : Int := 999;   // Номер последнего DB для PID-регулятора
   END_VAR
BEGIN
END_DATA_BLOCK

ORGANIZATION_BLOCK "Main"   // OB1, LAD, ProgramCycle
TITLE = "Main Program Sweep (Cycle)"
{ S7_Optimized_Access := 'TRUE' }
VERSION : 0.1
// stored: AutoNumber true, IsIECCheckEnabled false, SetENOAutomatically false
   VAR_INPUT
      Initial_Call : Bool;   // Initial call of this OB
      Remanence : Bool;   // =True, if remanent data are available
   END_VAR
   VAR_TEMP   // added for the SCL form of the ladder/FBD networks
      _w1 : Bool;
      _w2 : Bool;
   END_VAR
BEGIN

REGION Network 1
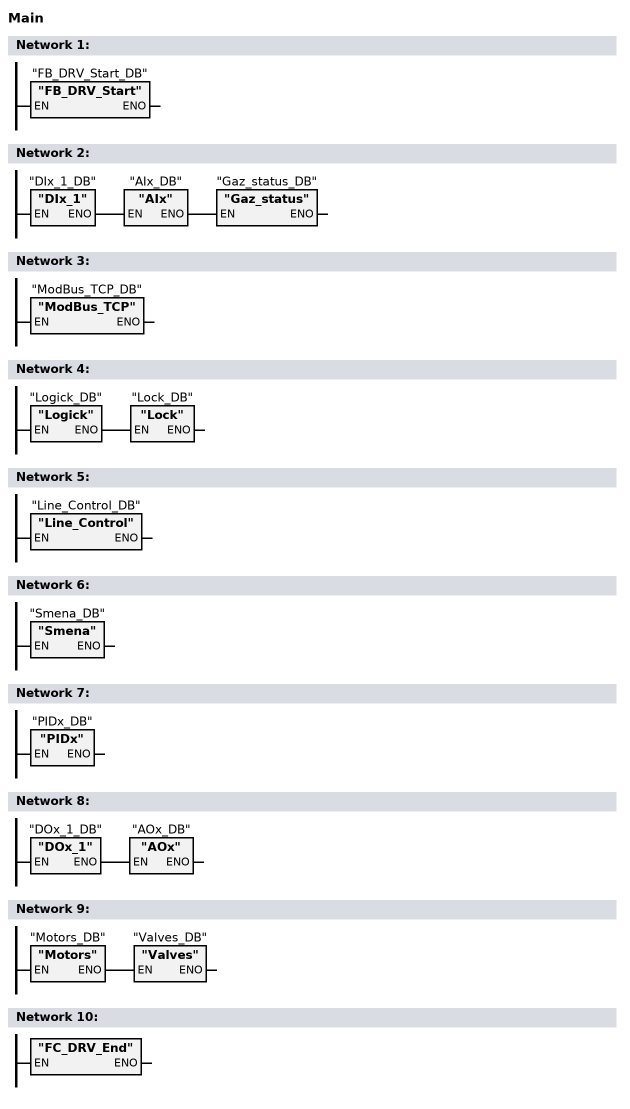
   RUNG wire#powerrail
      "FB_DRV_Start_DB"()
   END_RUNG
   // the same network as SCL:
   "FB_DRV_Start_DB"();   // "FB_DRV_Start"
END_REGION

REGION Network 2
   RUNG wire#powerrail
      "DIx_1_DB"()
      "AIx_DB"()
      "Gaz_status_DB"()
   END_RUNG
   // the same network as SCL:
   "DIx_1_DB"(ENO => #_w1);   // "DIx_1"
   "AIx_DB"(EN := #_w1, ENO => #_w2);   // "AIx"
   IF #_w2 THEN
       "Gaz_status_DB"();   // "Gaz_status"
   END_IF;
END_REGION

REGION Network 3
   RUNG wire#powerrail
      "ModBus_TCP_DB"()
   END_RUNG
   // the same network as SCL:
   "ModBus_TCP_DB"();   // "ModBus_TCP"
END_REGION

REGION Network 4
   RUNG wire#powerrail
      "Logick_DB"()
      "Lock_DB"()
   END_RUNG
   // the same network as SCL:
   "Logick_DB"(ENO => #_w1);   // "Logick"
   IF #_w1 THEN
       "Lock_DB"();   // "Lock"
   END_IF;
END_REGION

REGION Network 5
   RUNG wire#powerrail
      "Line_Control_DB"()
   END_RUNG
   // the same network as SCL:
   "Line_Control_DB"();   // "Line_Control"
END_REGION

REGION Network 6
   RUNG wire#powerrail
      "Smena_DB"()
   END_RUNG
   // the same network as SCL:
   "Smena_DB"();   // "Smena"
END_REGION

REGION Network 7
   RUNG wire#powerrail
      "PIDx_DB"()
   END_RUNG
   // the same network as SCL:
   "PIDx_DB"();   // "PIDx"
END_REGION

REGION Network 8
   RUNG wire#powerrail
      "DOx_1_DB"()
      "AOx_DB"()
   END_RUNG
   // the same network as SCL:
   "DOx_1_DB"(ENO => #_w1);   // "DOx_1"
   IF #_w1 THEN
       "AOx_DB"();   // "AOx"
   END_IF;
END_REGION

REGION Network 9
   RUNG wire#powerrail
      "Motors_DB"()
      "Valves_DB"()
   END_RUNG
   // the same network as SCL:
   "Motors_DB"(ENO => #_w1);   // "Motors"
   IF #_w1 THEN
       "Valves_DB"();   // "Valves"
   END_IF;
END_REGION

REGION Network 10
   RUNG wire#powerrail
      "FC_DRV_End"()
   END_RUNG
   // the same network as SCL:
   "FC_DRV_End"();
END_REGION
END_ORGANIZATION_BLOCK

FUNCTION_BLOCK "FB_DRV_Start"   // FB100, LAD
{ S7_Optimized_Access := 'TRUE' }
VERSION : 0.1
// stored: AutoNumber false, IsIECCheckEnabled false, IsRetainMemResEnabled false, MemoryReserve 100, SetENOAutomatically false, UDAEnableTagReadback false
   VAR
      last_01s : Int;
      last_05s : Int;
      last_1s : Int;
      last_5s : Int;
      last_10s : Int;
      last_30s : Int;
      last_1m : Int;
      last_5m : Int;
      last_10m : Int;
      last_30m : Int;
      last_1h : Int;
      last_1_day : Int;
      last_1_week : Int;
      last_1_month : Int;
      last_s1 : Int;
      last_s2 : Int;
      "1h_minutes" { S7_SetPoint := 'True'} : Int;
      "1_day_hour" { S7_SetPoint := 'True'} : Int;
      "1_day_minutes" { S7_SetPoint := 'True'} : Int;
      "1_week_weekday" { S7_SetPoint := 'True'} : Int := 1;
      "1_week_hour" { S7_SetPoint := 'True'} : Int;
      "1_week_minutes" { S7_SetPoint := 'True'} : Int;
      "1_month_date" { S7_SetPoint := 'True'} : Int := 1;
      "1_month_hour" { S7_SetPoint := 'True'} : Int;
      "1_month_minutes" { S7_SetPoint := 'True'} : Int;
      s1_hour : Int := 8;
      s1_minutes : Int;
      s2_hour : Int := 20;
      s2_minutes : Int;
      pos : Array[0..15] of Bool;
      Error : Word;
      x { S7_SetPoint := 'True'} : "Protection";
   END_VAR
   VAR_TEMP
      cnt_01s : Int;
      cnt_5s : Int;
      cnt_10s : Int;
      cnt_30s : Int;
      cnt_5m : Int;
      cnt_10m : Int;
      cnt_30m : Int;
   END_VAR
   VAR_TEMP   // added for the SCL form of the ladder/FBD networks
      _w1 : Bool;
      _w2 : Bool;
   END_VAR
BEGIN

REGION Network 1: Обработчик системного времени
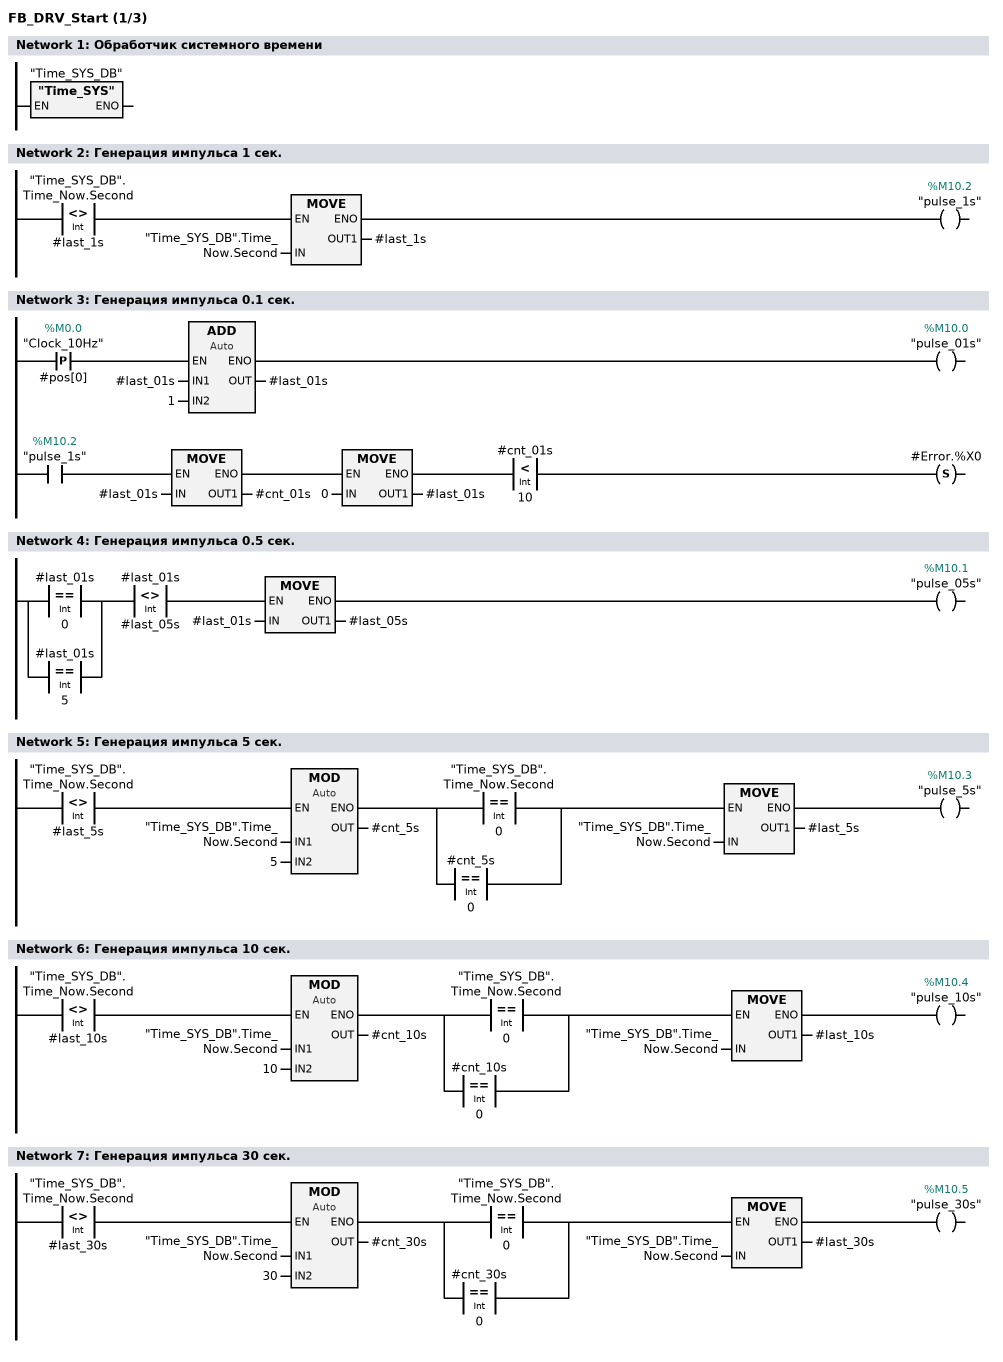
   RUNG wire#powerrail
      "Time_SYS_DB"()
   END_RUNG
   // the same network as SCL:
   "Time_SYS_DB"();   // "Time_SYS"
END_REGION

REGION Network 2: Генерация импульса 1 сек.
   RUNG wire#powerrail
      { S7_Templates := "SrcType := Int" } NE_Contact(in1 := "Time_SYS_DB".Time_Now.Second, in2 := #last_1s)
      Move(in := "Time_SYS_DB".Time_Now.Second, out1 => #last_1s)
      Coil( "pulse_1s" )
   END_RUNG
   // the same network as SCL:
   #_w1 := "Time_SYS_DB".Time_Now.Second <> #last_1s;
   IF #_w1 THEN #last_1s := "Time_SYS_DB".Time_Now.Second; END_IF;
   "pulse_1s" := #_w1;
END_REGION

REGION Network 3: Генерация импульса 0.1 сек.
   RUNG wire#powerrail
      P_Contact(operand := "Clock_10Hz", bit := #pos[0])
      Add(in1 := #last_01s, in2 := 1, out => #last_01s)
      Coil( "pulse_01s" )
   END_RUNG
   RUNG wire#powerrail
      Contact( "pulse_1s" )
      Move(in := #last_01s, out1 => #cnt_01s)
      Move(in := 0, out1 => #last_01s)
      { S7_Templates := "SrcType := Int" } LT_Contact(in1 := #cnt_01s, in2 := 10)
      S_Coil( #Error.%X0 )
   END_RUNG
   // the same network as SCL:
   #_w1 := "Clock_10Hz" AND NOT #pos[0];   // rising edge of "Clock_10Hz"
   #pos[0] := "Clock_10Hz";
   IF #_w1 THEN #last_01s := #last_01s + 1; END_IF;
   "pulse_01s" := #_w1;
   IF "pulse_1s" THEN
       #cnt_01s := #last_01s;
       #last_01s := 0;
   END_IF;
   IF "pulse_1s" AND (#cnt_01s < 10) THEN #Error.%X0 := TRUE; END_IF;
END_REGION

REGION Network 4: Генерация импульса 0.5 сек.
   RUNG wire#powerrail
      { S7_Templates := "SrcType := Int" } EQ_Contact(in1 := #last_01s, in2 := 0)
      wire#w1
      { S7_Templates := "SrcType := Int" } NE_Contact(in1 := #last_01s, in2 := #last_05s)
      Move(in := #last_01s, out1 => #last_05s)
      Coil( "pulse_05s" )
   END_RUNG
   RUNG wire#powerrail
      { S7_Templates := "SrcType := Int" } EQ_Contact(in1 := #last_01s, in2 := 5)
   END_RUNG wire#w1
   // the same network as SCL:
   #_w1 := ((#last_01s = 0) OR (#last_01s = 5)) AND (#last_01s <> #last_05s);
   IF #_w1 THEN #last_05s := #last_01s; END_IF;
   "pulse_05s" := #_w1;
END_REGION

REGION Network 5: Генерация импульса 5 сек.
   RUNG wire#powerrail
      { S7_Templates := "SrcType := Int" } NE_Contact(in1 := "Time_SYS_DB".Time_Now.Second, in2 := #last_5s)
      Mod(in1 := "Time_SYS_DB".Time_Now.Second, in2 := 5, out => #cnt_5s)
      wire#w1
      { S7_Templates := "SrcType := Int" } EQ_Contact(in1 := "Time_SYS_DB".Time_Now.Second, in2 := 0)
      wire#w2
      Move(in := "Time_SYS_DB".Time_Now.Second, out1 => #last_5s)
      Coil( "pulse_5s" )
   END_RUNG
   RUNG wire#w1
      { S7_Templates := "SrcType := Int" } EQ_Contact(in1 := #cnt_5s, in2 := 0)
   END_RUNG wire#w2
   // the same network as SCL:
   #_w1 := "Time_SYS_DB".Time_Now.Second <> #last_5s;
   IF #_w1 THEN #cnt_5s := "Time_SYS_DB".Time_Now.Second MOD 5; END_IF;
   #_w2 := #_w1 AND (("Time_SYS_DB".Time_Now.Second = 0) OR (#cnt_5s = 0));
   IF #_w2 THEN #last_5s := "Time_SYS_DB".Time_Now.Second; END_IF;
   "pulse_5s" := #_w2;
END_REGION

